# B&R Automation Studio project NAINV104C00R8L515F00 (part 5)

#### fHermesParseBoardAvailable.st
```iecst
(* Hermes Parse XML Table Data For Board Available *)
FUNCTION fHermesParseBoardAvailable

	fHermesParseBoardAvailable	:= TRUE;

	IF (tyXMLTableCurr.sTitle = 'AT') AND (sCurrValueLowerCase = 'boardid') THEN

		p_tyBoardAvailable.tyAvl.bBoardId	:= TRUE;

		IF tyXMLTableNxt.sTitle = 'AV' THEN
			p_tyBoardAvailable.tyData.sBoardId	:= tyXMLTableNxt.sValue;
		END_IF

	ELSIF (tyXMLTableCurr.sTitle = 'AT') AND (sCurrValueLowerCase = 'boardidcreatedby') THEN

		p_tyBoardAvailable.tyAvl.bBoardIdCreatedBy	:= TRUE;

		IF tyXMLTableNxt.sTitle = 'AV' THEN
			p_tyBoardAvailable.tyData.sBoardIdCreatedBy	:= tyXMLTableNxt.sValue;
		END_IF

	ELSIF (tyXMLTableCurr.sTitle = 'AT') AND (sCurrValueLowerCase = 'failedboard') THEN

		p_tyBoardAvailable.tyAvl.bFailedBoard	:= TRUE;

		IF tyXMLTableNxt.sTitle = 'AV' THEN
			IF tyXMLTableNxt.sValue = '1' THEN
				p_tyBoardAvailable.tyData.eFailedBoard	:= HermesGoodBoard;
			ELSIF tyXMLTableNxt.sValue = '2' THEN
				p_tyBoardAvailable.tyData.eFailedBoard	:= HermesFailedBoard;
			ELSE
				p_tyBoardAvailable.tyData.eFailedBoard	:= HermesUnknownBoard;
			END_IF
		END_IF

	ELSIF (tyXMLTableCurr.sTitle = 'AT') AND (sCurrValueLowerCase = 'producttypeid') THEN

		p_tyBoardAvailable.tyAvl.bProductTypeId	:= TRUE;

		IF tyXMLTableNxt.sTitle = 'AV' THEN
			p_tyBoardAvailable.tyData.sProductTypeId	:= tyXMLTableNxt.sValue;
		END_IF

	ELSIF (tyXMLTableCurr.sTitle = 'AT') AND (sCurrValueLowerCase = 'flippedboard') THEN

		p_tyBoardAvailable.tyAvl.bFlippedBoard	:= TRUE;

		IF tyXMLTableNxt.sTitle = 'AV' THEN
			IF tyXMLTableNxt.sValue = '1' THEN
				p_tyBoardAvailable.tyData.eFlippedBoard	:= HermesFlippedBoardTopSideUp;
			ELSIF tyXMLTableNxt.sValue = '2' THEN
				p_tyBoardAvailable.tyData.eFlippedBoard	:= HermesFlippedBoardBtmSideUp;
			ELSE
				p_tyBoardAvailable.tyData.eFlippedBoard	:= HermesFlippedBoardUnknownSide;
			END_IF
		END_IF

	ELSIF (tyXMLTableCurr.sTitle = 'AT') AND (sCurrValueLowerCase = 'topbarcode') THEN

		p_tyBoardAvailable.tyAvl.bTopBarcode	:= TRUE;

		IF tyXMLTableNxt.sTitle = 'AV' THEN
			p_tyBoardAvailable.tyData.sTopBarcode	:= tyXMLTableNxt.sValue;
		END_IF

	ELSIF (tyXMLTableCurr.sTitle = 'AT') AND (sCurrValueLowerCase = 'bottombarcode') THEN

		p_tyBoardAvailable.tyAvl.bBottomBarcode	:= TRUE;

		IF tyXMLTableNxt.sTitle = 'AV' THEN
			p_tyBoardAvailable.tyData.sBottomBarcode	:= tyXMLTableNxt.sValue;
		END_IF

	ELSIF (tyXMLTableCurr.sTitle = 'AT') AND (sCurrValueLowerCase = 'length') THEN

		p_tyBoardAvailable.tyAvl.bLength	:= TRUE;

		IF tyXMLTableNxt.sTitle = 'AV' THEN
			p_tyBoardAvailable.tyData.rLength	:= STRING_TO_REAL(tyXMLTableNxt.sValue);
		END_IF

	ELSIF (tyXMLTableCurr.sTitle = 'AT') AND (sCurrValueLowerCase = 'width') THEN

		p_tyBoardAvailable.tyAvl.bWidth	:= TRUE;

		IF tyXMLTableNxt.sTitle = 'AV' THEN
			p_tyBoardAvailable.tyData.rWidth	:= STRING_TO_REAL(tyXMLTableNxt.sValue);
		END_IF

	ELSIF (tyXMLTableCurr.sTitle = 'AT') AND (sCurrValueLowerCase = 'thickness') THEN

		p_tyBoardAvailable.tyAvl.bThickness	:= TRUE;

		IF tyXMLTableNxt.sTitle = 'AV' THEN
			p_tyBoardAvailable.tyData.rThickness	:= STRING_TO_REAL(tyXMLTableNxt.sValue);
		END_IF

	ELSIF (tyXMLTableCurr.sTitle = 'AT') AND (sCurrValueLowerCase = 'conveyorspeed') THEN

		p_tyBoardAvailable.tyAvl.bConveyorSpeed	:= TRUE;

		IF tyXMLTableNxt.sTitle = 'AV' THEN
			p_tyBoardAvailable.tyData.rConveyorSpeed	:= STRING_TO_REAL(tyXMLTableNxt.sValue);
		END_IF

	ELSIF (tyXMLTableCurr.sTitle = 'AT') AND (sCurrValueLowerCase = 'topclearanceheight') THEN

		p_tyBoardAvailable.tyAvl.bTopClearanceHeight	:= TRUE;

		IF tyXMLTableNxt.sTitle = 'AV' THEN
			p_tyBoardAvailable.tyData.rTopClearanceHeight	:= STRING_TO_REAL(tyXMLTableNxt.sValue);
		END_IF

	ELSIF (tyXMLTableCurr.sTitle = 'AT') AND (sCurrValueLowerCase = 'bottomclearanceheight') THEN

		p_tyBoardAvailable.tyAvl.bBottomClearanceHeight	:= TRUE;

		IF tyXMLTableNxt.sTitle = 'AV' THEN
			p_tyBoardAvailable.tyData.rBottomClearanceHeight	:= STRING_TO_REAL(tyXMLTableNxt.sValue);
		END_IF

	ELSIF (tyXMLTableCurr.sTitle = 'AT') AND (sCurrValueLowerCase = 'weight') THEN

		p_tyBoardAvailable.tyAvl.bWeight	:= TRUE;

		IF tyXMLTableNxt.sTitle = 'AV' THEN
			p_tyBoardAvailable.tyData.rWeight	:= STRING_TO_REAL(tyXMLTableNxt.sValue);
		END_IF

	ELSIF (tyXMLTableCurr.sTitle = 'AT') AND (sCurrValueLowerCase = 'workorderid') THEN

		p_tyBoardAvailable.tyAvl.bWorkOrderId	:= TRUE;

		IF tyXMLTableNxt.sTitle = 'AV' THEN
			p_tyBoardAvailable.tyData.sWorkOrderId	:= tyXMLTableNxt.sValue;
		END_IF

	ELSIF (tyXMLTableCurr.sTitle = 'AT') AND (sCurrValueLowerCase = 'batchid') THEN

		p_tyBoardAvailable.tyAvl.bBatchId	:= TRUE;

		IF tyXMLTableNxt.sTitle = 'AV' THEN
			p_tyBoardAvailable.tyData.sBatchId	:= tyXMLTableNxt.sValue;
		END_IF
	ELSIF (tyXMLTableCurr.sTitle = 'AT') AND (sCurrValueLowerCase = 'route') THEN

		p_tyBoardAvailable.tyAvl.bRoute	:= TRUE;

		IF tyXMLTableNxt.sTitle = 'AV' THEN
			p_tyBoardAvailable.tyData.iRoute	:= STRING_TO_INT(tyXMLTableNxt.sValue);
		END_IF
	ELSIF (tyXMLTableCurr.sTitle = 'AT') AND (sCurrValueLowerCase = 'action') THEN

		p_tyBoardAvailable.tyAvl.bAction	:= TRUE;

		IF tyXMLTableNxt.sTitle = 'AV' THEN
			p_tyBoardAvailable.tyData.iAction	:= STRING_TO_INT(tyXMLTableNxt.sValue);
		END_IF
	ELSIF (tyXMLTableCurr.sTitle = 'ST') AND (sCurrValueLowerCase = 'sb') THEN
		iSubBoardCntr := iSubBoardCntr + 1;
	ELSIF (tyXMLTableCurr.sTitle = 'AT') AND (sCurrValueLowerCase = 'pos') THEN
		p_tyBoardAvailable.tyAvl.tySubBoards.bSubBoardsPos[iSubBoardCntr]	:= TRUE;

		IF tyXMLTableNxt.sTitle = 'AV' THEN
			p_tyBoardAvailable.tyData.tySubBoards.iSubBoardsPos[iSubBoardCntr]	:= STRING_TO_INT(tyXMLTableNxt.sValue);
		END_IF
	ELSIF (tyXMLTableCurr.sTitle = 'AT') AND (sCurrValueLowerCase = 'bc') THEN

		p_tyBoardAvailable.tyAvl.tySubBoards.bSubBoardsBc[iSubBoardCntr]	:= TRUE;

		IF tyXMLTableNxt.sTitle = 'AV' THEN
			p_tyBoardAvailable.tyData.tySubBoards.sSubBoardsBc[iSubBoardCntr]	:= tyXMLTableNxt.sValue;
		END_IF
	ELSIF (tyXMLTableCurr.sTitle = 'AT') AND (sCurrValueLowerCase = 'st') THEN

		p_tyBoardAvailable.tyAvl.tySubBoards.bSubBoardsSt[iSubBoardCntr]	:= TRUE;

		IF tyXMLTableNxt.sTitle = 'AV' THEN
			p_tyBoardAvailable.tyData.tySubBoards.iSubBoardsSt[iSubBoardCntr]	:= STRING_TO_INT(tyXMLTableNxt.sValue);
		END_IF
	END_IF

END_FUNCTION
```

#### fHermesParseMachineReady.st
```iecst
(* Hermes Parse XML Table Data For Machine Ready*)
FUNCTION fHermesParseMachineReady

	fHermesParseMachineReady	:= TRUE;

	IF (tyXMLTableCurr.sTitle = 'AT') AND (sCurrValueLowerCase = 'failedboard') THEN

		p_tyMachineReady.tyAvl.bFailedBoard	:= TRUE;

		IF tyXMLTableNxt.sTitle = 'AV' THEN
			IF tyXMLTableNxt.sValue = '1' THEN
				p_tyMachineReady.tyData.eFailedBoard	:= HermesGoodBoard;
			ELSIF tyXMLTableNxt.sValue = '2' THEN
				p_tyMachineReady.tyData.eFailedBoard	:= HermesFailedBoard;
			ELSE
				p_tyMachineReady.tyData.eFailedBoard	:= HermesUnknownBoard;
			END_IF
		END_IF

	ELSIF (tyXMLTableCurr.sTitle = 'AT') AND (sCurrValueLowerCase = 'forecastid') THEN

		p_tyMachineReady.tyAvl.bForecastId	:= TRUE;

		IF tyXMLTableNxt.sTitle = 'AV' THEN
			p_tyMachineReady.tyData.sForecastId	:= tyXMLTableNxt.sValue;
		END_IF

	ELSIF (tyXMLTableCurr.sTitle = 'AT') AND (sCurrValueLowerCase = 'boardid') THEN

		p_tyMachineReady.tyAvl.bBoardId	:= TRUE;

		IF tyXMLTableNxt.sTitle = 'AV' THEN
			p_tyMachineReady.tyData.sBoardId	:= tyXMLTableNxt.sValue;
		END_IF

	ELSIF (tyXMLTableCurr.sTitle = 'AT') AND (sCurrValueLowerCase = 'producttypeid') THEN

		p_tyMachineReady.tyAvl.bProductTypeId	:= TRUE;

		IF tyXMLTableNxt.sTitle = 'AV' THEN
			p_tyMachineReady.tyData.sProductTypeId	:= tyXMLTableNxt.sValue;
		END_IF

	ELSIF (tyXMLTableCurr.sTitle = 'AT') AND (sCurrValueLowerCase = 'flippedboard') THEN

		p_tyMachineReady.tyAvl.bFlippedBoard	:= TRUE;

		IF tyXMLTableNxt.sTitle = 'AV' THEN
			IF tyXMLTableNxt.sValue = '1' THEN
				p_tyMachineReady.tyData.eFlippedBoard	:= HermesFlippedBoardTopSideUp;
			ELSIF tyXMLTableNxt.sValue = '2' THEN
				p_tyMachineReady.tyData.eFlippedBoard	:= HermesFlippedBoardBtmSideUp;
			ELSE
				p_tyMachineReady.tyData.eFlippedBoard	:= HermesFlippedBoardUnknownSide;
			END_IF
		END_IF

	ELSIF (tyXMLTableCurr.sTitle = 'AT') AND (sCurrValueLowerCase = 'length') THEN

		p_tyMachineReady.tyAvl.bLength	:= TRUE;

		IF tyXMLTableNxt.sTitle = 'AV' THEN
			p_tyMachineReady.tyData.rLength	:= STRING_TO_REAL(tyXMLTableNxt.sValue);
		END_IF

	ELSIF (tyXMLTableCurr.sTitle = 'AT') AND (sCurrValueLowerCase = 'width') THEN

		p_tyMachineReady.tyAvl.bWidth	:= TRUE;

		IF tyXMLTableNxt.sTitle = 'AV' THEN
			p_tyMachineReady.tyData.rWidth	:= STRING_TO_REAL(tyXMLTableNxt.sValue);
		END_IF

	ELSIF (tyXMLTableCurr.sTitle = 'AT') AND (sCurrValueLowerCase = 'thickness') THEN

		p_tyMachineReady.tyAvl.bThickness	:= TRUE;

		IF tyXMLTableNxt.sTitle = 'AV' THEN
			p_tyMachineReady.tyData.rThickness	:= STRING_TO_REAL(tyXMLTableNxt.sValue);
		END_IF

	ELSIF (tyXMLTableCurr.sTitle = 'AT') AND (sCurrValueLowerCase = 'conveyorspeed') THEN

		p_tyMachineReady.tyAvl.bConveyorSpeed	:= TRUE;

		IF tyXMLTableNxt.sTitle = 'AV' THEN
			p_tyMachineReady.tyData.rConveyorSpeed	:= STRING_TO_REAL(tyXMLTableNxt.sValue);
		END_IF

	ELSIF (tyXMLTableCurr.sTitle = 'AT') AND (sCurrValueLowerCase = 'topclearanceheight') THEN

		p_tyMachineReady.tyAvl.bTopClearanceHeight	:= TRUE;

		IF tyXMLTableNxt.sTitle = 'AV' THEN
			p_tyMachineReady.tyData.rTopClearanceHeight	:= STRING_TO_REAL(tyXMLTableNxt.sValue);
		END_IF

	ELSIF (tyXMLTableCurr.sTitle = 'AT') AND (sCurrValueLowerCase = 'bottomclearanceheight') THEN

		p_tyMachineReady.tyAvl.bBottomClearanceHeight	:= TRUE;

		IF tyXMLTableNxt.sTitle = 'AV' THEN
			p_tyMachineReady.tyData.rBottomClearanceHeight	:= STRING_TO_REAL(tyXMLTableNxt.sValue);
		END_IF

	ELSIF (tyXMLTableCurr.sTitle = 'AT') AND (sCurrValueLowerCase = 'weight') THEN

		p_tyMachineReady.tyAvl.bWeight	:= TRUE;

		IF tyXMLTableNxt.sTitle = 'AV' THEN
			p_tyMachineReady.tyData.rWeight	:= STRING_TO_REAL(tyXMLTableNxt.sValue);
		END_IF

	ELSIF (tyXMLTableCurr.sTitle = 'AT') AND (sCurrValueLowerCase = 'workorderid') THEN

		p_tyMachineReady.tyAvl.bWorkOrderId	:= TRUE;

		IF tyXMLTableNxt.sTitle = 'AV' THEN
			p_tyMachineReady.tyData.sWorkOrderId	:= tyXMLTableNxt.sValue;
		END_IF

	ELSIF (tyXMLTableCurr.sTitle = 'AT') AND (sCurrValueLowerCase = 'batchid') THEN

		p_tyMachineReady.tyAvl.bBatchId	:= TRUE;

		IF tyXMLTableNxt.sTitle = 'AV' THEN
			p_tyMachineReady.tyData.sBatchId	:= tyXMLTableNxt.sValue;
		END_IF

	END_IF

END_FUNCTION
```

#### fHermesParseStartTransport.st
```iecst
(* Hermes Parse XML Table Data For Start Transport*)
FUNCTION fHermesParseStartTransport

	fHermesParseStartTransport	:= TRUE;

	IF (tyXMLTableCurr.sTitle = 'AT') AND (sCurrValueLowerCase = 'boardid') THEN

		p_tyStartTransport.tyAvl.bBoardId	:= TRUE;

		IF tyXMLTableNxt.sTitle = 'AV' THEN
			p_tyStartTransport.tyData.sBoardId	:= tyXMLTableNxt.sValue;
		END_IF

	ELSIF (tyXMLTableCurr.sTitle = 'AT') AND (sCurrValueLowerCase = 'conveyorspeed') THEN

		p_tyStartTransport.tyAvl.bConveyorSpeed	:= TRUE;

		IF tyXMLTableNxt.sTitle = 'AV' THEN
			p_tyStartTransport.tyData.rConveyorSpeed	:= STRING_TO_REAL(tyXMLTableNxt.sValue);
		END_IF

	END_IF

END_FUNCTION
```

#### fHermesParseStopTransport.st
```iecst
(* Hermes Parse XML Table Data For Stop Transport*)
FUNCTION fHermesParseStopTransport

	fHermesParseStopTransport	:= TRUE;

	IF (tyXMLTableCurr.sTitle = 'AT') AND (sCurrValueLowerCase = 'transferstate') THEN

		p_tyStopTransport.tyAvl.bTransferState	:= TRUE;

		IF tyXMLTableNxt.sTitle = 'AV' THEN
			IF tyXMLTableNxt.sValue = '1' THEN
				p_tyStopTransport.tyData.eTransferState	:= HermesTransferStateNotStarted;
			ELSIF tyXMLTableNxt.sValue = '2' THEN
				p_tyStopTransport.tyData.eTransferState	:= HermesTransferStateIncomplete;
			ELSE
				p_tyStopTransport.tyData.eTransferState	:= HermesTransferStateComplete;
			END_IF
		END_IF

	ELSIF (tyXMLTableCurr.sTitle = 'AT') AND (sCurrValueLowerCase = 'boardid') THEN

		p_tyStopTransport.tyAvl.bBoardId	:= TRUE;

		IF tyXMLTableNxt.sTitle = 'AV' THEN
			p_tyStopTransport.tyData.sBoardId	:= tyXMLTableNxt.sValue;
		END_IF

	END_IF

END_FUNCTION
```

#### fHermesParseTransportFinished.st
```iecst
(* Hermes Parse XML Table Data For Transport Finished *)
FUNCTION fHermesParseTransportFinished

	fHermesParseTransportFinished	:= TRUE;

	IF (tyXMLTableCurr.sTitle = 'AT') AND (sCurrValueLowerCase = 'transferstate') THEN

		p_tyTransportFinished.tyAvl.bTransferState	:= TRUE;

		IF tyXMLTableNxt.sTitle = 'AV' THEN
			IF tyXMLTableNxt.sValue = '1' THEN
				p_tyTransportFinished.tyData.eTransferState	:= HermesTransferStateNotStarted;
			ELSIF tyXMLTableNxt.sValue = '2' THEN
				p_tyTransportFinished.tyData.eTransferState	:= HermesTransferStateIncomplete;
			ELSE
				p_tyTransportFinished.tyData.eTransferState	:= HermesTransferStateComplete;
			END_IF
		END_IF

	ELSIF (tyXMLTableCurr.sTitle = 'AT') AND (sCurrValueLowerCase = 'boardid') THEN

		p_tyTransportFinished.tyAvl.bBoardId	:= TRUE;

		IF tyXMLTableNxt.sTitle = 'AV' THEN
			p_tyTransportFinished.tyData.sBoardId	:= tyXMLTableNxt.sValue;
		END_IF

	END_IF

END_FUNCTION
```

#### fHermesParseSetConfiguration.st
```iecst
(* Hermes Parse XML Table Data For Set Configuration*)
FUNCTION fHermesParseSetConfiguration

	fHermesParseSetConfiguration	:= TRUE;

	IF (tyXMLTableCurr.sTitle = 'AT') AND (sCurrValueLowerCase = 'machineid') THEN

		p_tySetConfiguration.tyAvl.bMachineId	:= TRUE;

		IF tyXMLTableNxt.sTitle = 'AV' THEN
			p_tySetConfiguration.tyData.sMachineId	:= tyXMLTableNxt.sValue;
		END_IF

	ELSIF (tyXMLTableCurr.sTitle = 'AT') AND (sCurrValueLowerCase = 'supervisorysystemport') THEN

		p_tySetConfiguration.tyAvl.bSupervisorySystemPort	:= TRUE;

		IF tyXMLTableNxt.sTitle = 'AV' THEN
			p_tySetConfiguration.tyData.uiSupervisorySystemPort	:= STRING_TO_UINT(tyXMLTableNxt.sValue);
		END_IF

	ELSIF (tyXMLTableCurr.sTitle = 'ST') AND (sCurrValueLowerCase = 'upstreamconfigurations') THEN

		bUpstream	:= TRUE;
		bDownstream	:= FALSE;

	ELSIF (tyXMLTableCurr.sTitle = 'ET') AND (sCurrValueLowerCase = 'upstreamconfigurations') THEN

		bUpstream	:= FALSE;

	ELSIF (tyXMLTableCurr.sTitle = 'ST') AND (sCurrValueLowerCase = 'downstreamconfigurations') THEN

		bUpstream	:= FALSE;
		bDownstream	:= TRUE;

	ELSIF (tyXMLTableCurr.sTitle = 'ET') AND (sCurrValueLowerCase = 'downstreamconfigurations') THEN

		bDownstream	:= FALSE;

	ELSIF bUpstream = TRUE THEN

		IF (tyXMLTableCurr.sTitle = 'ST') AND (sCurrValueLowerCase = 'upstreamconfiguration') THEN

			p_tySetConfiguration.tyAvl.bUpstreamConfigurations	:= TRUE;

			p_tySetConfiguration.tyAvl.iUpstreamConfigurations	:= p_tySetConfiguration.tyAvl.iUpstreamConfigurations + 1;
//			IF p_tySetConfiguration.tyAvl.iUpstreamConfigurations > 3 THEN
//				p_tySetConfiguration.tyAvl.iUpstreamConfigurations	:= 3;
//			END_IF

		ELSIF p_tySetConfiguration.tyAvl.iUpstreamConfigurations <> 0 THEN

			IF (tyXMLTableCurr.sTitle = 'AT') AND (sCurrValueLowerCase = 'upstreamlaneid') THEN

				p_tySetConfiguration.tyAvl.a_tyUpstreamConfigurations[p_tySetConfiguration.tyAvl.iUpstreamConfigurations - 1].bUpstreamLaneId	:= TRUE;

				IF tyXMLTableNxt.sTitle = 'AV' THEN
					p_tySetConfiguration.tyData.a_tyUpstreamConfigurations[p_tySetConfiguration.tyAvl.iUpstreamConfigurations - 1].iUpstreamLaneId	:= STRING_TO_INT(tyXMLTableNxt.sValue);
				END_IF

			ELSIF (tyXMLTableCurr.sTitle = 'AT') AND (sCurrValueLowerCase = 'upstreaminterfaceid') THEN

				p_tySetConfiguration.tyAvl.a_tyUpstreamConfigurations[p_tySetConfiguration.tyAvl.iUpstreamConfigurations - 1].bUpstreamInterfaceId	:= TRUE;

				IF tyXMLTableNxt.sTitle = 'AV' THEN
					p_tySetConfiguration.tyData.a_tyUpstreamConfigurations[p_tySetConfiguration.tyAvl.iUpstreamConfigurations - 1].sUpstreamInterfaceId	:= tyXMLTableNxt.sValue;
				END_IF

			ELSIF (tyXMLTableCurr.sTitle = 'AT') AND (sCurrValueLowerCase = 'hostaddress') THEN

				p_tySetConfiguration.tyAvl.a_tyUpstreamConfigurations[p_tySetConfiguration.tyAvl.iUpstreamConfigurations - 1].bHostAddress	:= TRUE;

				IF tyXMLTableNxt.sTitle = 'AV' THEN
					p_tySetConfiguration.tyData.a_tyUpstreamConfigurations[p_tySetConfiguration.tyAvl.iUpstreamConfigurations - 1].sHostAddress	:= tyXMLTableNxt.sValue;
				END_IF

			ELSIF (tyXMLTableCurr.sTitle = 'AT') AND (sCurrValueLowerCase = 'port') THEN

				p_tySetConfiguration.tyAvl.a_tyUpstreamConfigurations[p_tySetConfiguration.tyAvl.iUpstreamConfigurations - 1].bPort	:= TRUE;

				IF tyXMLTableNxt.sTitle = 'AV' THEN
					p_tySetConfiguration.tyData.a_tyUpstreamConfigurations[p_tySetConfiguration.tyAvl.iUpstreamConfigurations - 1].uiPort	:= STRING_TO_UINT(tyXMLTableNxt.sValue);
				END_IF

			END_IF

		END_IF

	ELSIF bDownstream = TRUE THEN

		IF (tyXMLTableCurr.sTitle = 'ST') AND (sCurrValueLowerCase = 'downstreamconfiguration') THEN

			p_tySetConfiguration.tyAvl.bDownstreamConfigurations	:= TRUE;

			p_tySetConfiguration.tyAvl.iDownstreamConfigurations	:= p_tySetConfiguration.tyAvl.iDownstreamConfigurations + 1;
//			IF p_tySetConfiguration.tyAvl.iDownstreamConfigurations > 3 THEN
//				p_tySetConfiguration.tyAvl.iDownstreamConfigurations	:= 3;
//			END_IF

		ELSIF p_tySetConfiguration.tyAvl.iDownstreamConfigurations <> 0 THEN

			IF (tyXMLTableCurr.sTitle = 'AT') AND (sCurrValueLowerCase = 'downstreamlaneid') THEN

				p_tySetConfiguration.tyAvl.a_tyDownstreamConfigurations[p_tySetConfiguration.tyAvl.iDownstreamConfigurations - 1].bDownstreamLaneId	:= TRUE;

				IF tyXMLTableNxt.sTitle = 'AV' THEN
					p_tySetConfiguration.tyData.a_tyDownstreamConfigurations[p_tySetConfiguration.tyAvl.iDownstreamConfigurations - 1].iDownstreamLaneId	:= STRING_TO_INT(tyXMLTableNxt.sValue);
				END_IF

			ELSIF (tyXMLTableCurr.sTitle = 'AT') AND (sCurrValueLowerCase = 'downstreaminterfaceid') THEN

				p_tySetConfiguration.tyAvl.a_tyDownstreamConfigurations[p_tySetConfiguration.tyAvl.iDownstreamConfigurations - 1].bDownstreamInterfaceId	:= TRUE;

				IF tyXMLTableNxt.sTitle = 'AV' THEN
					p_tySetConfiguration.tyData.a_tyDownstreamConfigurations[p_tySetConfiguration.tyAvl.iDownstreamConfigurations - 1].sDownstreamInterfaceId	:= tyXMLTableNxt.sValue;
				END_IF

			ELSIF (tyXMLTableCurr.sTitle = 'AT') AND (sCurrValueLowerCase = 'clientaddress') THEN

				p_tySetConfiguration.tyAvl.a_tyDownstreamConfigurations[p_tySetConfiguration.tyAvl.iDownstreamConfigurations - 1].bClientAddress	:= TRUE;

				IF tyXMLTableNxt.sTitle = 'AV' THEN
					p_tySetConfiguration.tyData.a_tyDownstreamConfigurations[p_tySetConfiguration.tyAvl.iDownstreamConfigurations - 1].sClientAddress	:= tyXMLTableNxt.sValue;
				END_IF

			ELSIF (tyXMLTableCurr.sTitle = 'AT') AND (sCurrValueLowerCase = 'port') THEN

				p_tySetConfiguration.tyAvl.a_tyDownstreamConfigurations[p_tySetConfiguration.tyAvl.iDownstreamConfigurations - 1].bPort	:= TRUE;

				IF tyXMLTableNxt.sTitle = 'AV' THEN
					p_tySetConfiguration.tyData.a_tyDownstreamConfigurations[p_tySetConfiguration.tyAvl.iDownstreamConfigurations - 1].uiPort	:= STRING_TO_UINT(tyXMLTableNxt.sValue);
				END_IF

			END_IF

		END_IF

	END_IF

END_FUNCTION
```

#### fHermesParseCurrentConfiguration.st
```iecst
(* Hermes Parse XML Table Data For Current Configuration*)
FUNCTION fHermesParseCurrentConfiguration

	fHermesParseCurrentConfiguration	:= TRUE;

	IF (tyXMLTableCurr.sTitle = 'AT') AND (sCurrValueLowerCase = 'machineid') THEN

		p_tyCurrentConfiguration.tyAvl.bMachineId	:= TRUE;

		IF tyXMLTableNxt.sTitle = 'AV' THEN
			p_tyCurrentConfiguration.tyData.sMachineId	:= tyXMLTableNxt.sValue;
		END_IF

	ELSIF (tyXMLTableCurr.sTitle = 'AT') AND (sCurrValueLowerCase = 'supervisorysytemport') THEN

			p_tyCurrentConfiguration.tyAvl.bSupervisorySystemPort	:= TRUE;

			IF tyXMLTableNxt.sTitle = 'AV' THEN
				p_tyCurrentConfiguration.tyData.uiSupervisorySystemPort	:= STRING_TO_UINT(tyXMLTableNxt.sValue);
			END_IF

	ELSIF (tyXMLTableCurr.sTitle = 'ST') AND (sCurrValueLowerCase = 'upstreamconfigurations') THEN

		bUpstream	:= TRUE;
		bDownstream	:= FALSE;

	ELSIF (tyXMLTableCurr.sTitle = 'ET') AND (sCurrValueLowerCase = 'upstreamconfigurations') THEN

		bUpstream	:= FALSE;

	ELSIF (tyXMLTableCurr.sTitle = 'ST') AND (sCurrValueLowerCase = 'downstreamconfigurations') THEN

		bUpstream	:= FALSE;
		bDownstream	:= TRUE;

	ELSIF (tyXMLTableCurr.sTitle = 'ET') AND (sCurrValueLowerCase = 'downstreamconfigurations') THEN

		bDownstream	:= FALSE;

	ELSIF bUpstream = TRUE THEN

		IF (tyXMLTableCurr.sTitle = 'ST') AND (sCurrValueLowerCase = 'upstreamconfiguration') THEN

			p_tyCurrentConfiguration.tyAvl.bUpstreamConfigurations	:= TRUE;

			p_tyCurrentConfiguration.tyAvl.iUpstreamConfigurations	:= p_tyCurrentConfiguration.tyAvl.iUpstreamConfigurations + 1;
			IF p_tyCurrentConfiguration.tyAvl.iUpstreamConfigurations > 3 THEN
				p_tyCurrentConfiguration.tyAvl.iUpstreamConfigurations	:= 3;
			END_IF

		ELSIF p_tyCurrentConfiguration.tyAvl.iUpstreamConfigurations <> 0 THEN

			IF (tyXMLTableCurr.sTitle = 'AT') AND (sCurrValueLowerCase = 'upstreamlaneid') THEN

				p_tyCurrentConfiguration.tyAvl.a_tyUpstreamConfigurations[p_tyCurrentConfiguration.tyAvl.iUpstreamConfigurations - 1].bUpstreamLaneId	:= TRUE;

				IF tyXMLTableNxt.sTitle = 'AV' THEN
					p_tyCurrentConfiguration.tyData.a_tyUpstreamConfigurations[p_tyCurrentConfiguration.tyAvl.iUpstreamConfigurations - 1].iUpstreamLaneId	:= STRING_TO_INT(tyXMLTableNxt.sValue);
				END_IF

			ELSIF (tyXMLTableCurr.sTitle = 'AT') AND (sCurrValueLowerCase = 'upstreaminterfaceid') THEN

				p_tyCurrentConfiguration.tyAvl.a_tyUpstreamConfigurations[p_tyCurrentConfiguration.tyAvl.iUpstreamConfigurations - 1].bUpstreamInterfaceId	:= TRUE;

				IF tyXMLTableNxt.sTitle = 'AV' THEN
					p_tyCurrentConfiguration.tyData.a_tyUpstreamConfigurations[p_tyCurrentConfiguration.tyAvl.iUpstreamConfigurations - 1].sUpstreamInterfaceId	:= tyXMLTableNxt.sValue;
				END_IF

			ELSIF (tyXMLTableCurr.sTitle = 'AT') AND (sCurrValueLowerCase = 'hostaddress') THEN

				p_tyCurrentConfiguration.tyAvl.a_tyUpstreamConfigurations[p_tyCurrentConfiguration.tyAvl.iUpstreamConfigurations - 1].bHostAddress	:= TRUE;

				IF tyXMLTableNxt.sTitle = 'AV' THEN
					p_tyCurrentConfiguration.tyData.a_tyUpstreamConfigurations[p_tyCurrentConfiguration.tyAvl.iUpstreamConfigurations - 1].sHostAddress	:= tyXMLTableNxt.sValue;
				END_IF

			ELSIF (tyXMLTableCurr.sTitle = 'AT') AND (sCurrValueLowerCase = 'port') THEN

				p_tyCurrentConfiguration.tyAvl.a_tyUpstreamConfigurations[p_tyCurrentConfiguration.tyAvl.iUpstreamConfigurations - 1].bPort	:= TRUE;

				IF tyXMLTableNxt.sTitle = 'AV' THEN
					p_tyCurrentConfiguration.tyData.a_tyUpstreamConfigurations[p_tyCurrentConfiguration.tyAvl.iUpstreamConfigurations - 1].uiPort	:= STRING_TO_UINT(tyXMLTableNxt.sValue);
				END_IF

			END_IF

		END_IF

	ELSIF bDownstream = TRUE THEN

		IF (tyXMLTableCurr.sTitle = 'ST') AND (sCurrValueLowerCase = 'downstreamconfiguration') THEN

			p_tyCurrentConfiguration.tyAvl.bDownstreamConfigurations	:= TRUE;

			p_tyCurrentConfiguration.tyAvl.iDownstreamConfigurations	:= p_tyCurrentConfiguration.tyAvl.iDownstreamConfigurations + 1;
			IF p_tyCurrentConfiguration.tyAvl.iDownstreamConfigurations > 3 THEN
				p_tyCurrentConfiguration.tyAvl.iDownstreamConfigurations	:= 3;
			END_IF

		ELSIF p_tyCurrentConfiguration.tyAvl.iDownstreamConfigurations <> 0 THEN

			IF (tyXMLTableCurr.sTitle = 'AT') AND (sCurrValueLowerCase = 'downstreamlaneid') THEN

				p_tyCurrentConfiguration.tyAvl.a_tyDownstreamConfigurations[p_tyCurrentConfiguration.tyAvl.iDownstreamConfigurations - 1].bDownstreamLaneId	:= TRUE;

				IF tyXMLTableNxt.sTitle = 'AV' THEN
					p_tyCurrentConfiguration.tyData.a_tyDownstreamConfigurations[p_tyCurrentConfiguration.tyAvl.iDownstreamConfigurations - 1].iDownstreamLaneId	:= STRING_TO_INT(tyXMLTableNxt.sValue);
				END_IF

			ELSIF (tyXMLTableCurr.sTitle = 'AT') AND (sCurrValueLowerCase = 'downstreaminterfaceid') THEN

				p_tyCurrentConfiguration.tyAvl.a_tyDownstreamConfigurations[p_tyCurrentConfiguration.tyAvl.iDownstreamConfigurations - 1].bDownstreamInterfaceId	:= TRUE;

				IF tyXMLTableNxt.sTitle = 'AV' THEN
					p_tyCurrentConfiguration.tyData.a_tyDownstreamConfigurations[p_tyCurrentConfiguration.tyAvl.iDownstreamConfigurations - 1].sDownstreamInterfaceId	:= tyXMLTableNxt.sValue;
				END_IF

			ELSIF (tyXMLTableCurr.sTitle = 'AT') AND (sCurrValueLowerCase = 'clientaddress') THEN

				p_tyCurrentConfiguration.tyAvl.a_tyDownstreamConfigurations[p_tyCurrentConfiguration.tyAvl.iDownstreamConfigurations - 1].bClientAddress	:= TRUE;

				IF tyXMLTableNxt.sTitle = 'AV' THEN
					p_tyCurrentConfiguration.tyData.a_tyDownstreamConfigurations[p_tyCurrentConfiguration.tyAvl.iDownstreamConfigurations - 1].sClientAddress	:= tyXMLTableNxt.sValue;
				END_IF

			ELSIF (tyXMLTableCurr.sTitle = 'AT') AND (sCurrValueLowerCase = 'port') THEN

				p_tyCurrentConfiguration.tyAvl.a_tyDownstreamConfigurations[p_tyCurrentConfiguration.tyAvl.iDownstreamConfigurations - 1].bPort	:= TRUE;

				IF tyXMLTableNxt.sTitle = 'AV' THEN
					p_tyCurrentConfiguration.tyData.a_tyDownstreamConfigurations[p_tyCurrentConfiguration.tyAvl.iDownstreamConfigurations - 1].uiPort	:= STRING_TO_UINT(tyXMLTableNxt.sValue);
				END_IF

			END_IF

		END_IF

	END_IF

END_FUNCTION
```

#### fHermesParseBoardForecast.st
```iecst
(* Hermes Parse XML Table Data For Board Forecast*)
FUNCTION fHermesParseBoardForecast

	fHermesParseBoardForecast	:= TRUE;

	IF (tyXMLTableCurr.sTitle = 'AT') AND (sCurrValueLowerCase = 'forecastid') THEN

		p_tyBoardForecast.tyAvl.bForecastId	:= TRUE;

		IF tyXMLTableNxt.sTitle = 'AV' THEN
			p_tyBoardForecast.tyData.sForecastId	:= tyXMLTableNxt.sValue;
		END_IF

	ELSIF (tyXMLTableCurr.sTitle = 'AT') AND (sCurrValueLowerCase = 'timeuntilavailable') THEN

		p_tyBoardForecast.tyAvl.bTimeUntilAvailable	:= TRUE;

		IF tyXMLTableNxt.sTitle = 'AV' THEN
			p_tyBoardForecast.tyData.rTimeUntilAvailable	:= STRING_TO_REAL(tyXMLTableNxt.sValue);
		END_IF

	ELSIF (tyXMLTableCurr.sTitle = 'AT') AND (sCurrValueLowerCase = 'boardid') THEN

		p_tyBoardForecast.tyAvl.bBoardId	:= TRUE;

		IF tyXMLTableNxt.sTitle = 'AV' THEN
			p_tyBoardForecast.tyData.sBoardId	:= tyXMLTableNxt.sValue;
		END_IF

	ELSIF (tyXMLTableCurr.sTitle = 'AT') AND (sCurrValueLowerCase = 'boardidcreatedby') THEN

		p_tyBoardForecast.tyAvl.bBoardIdCreatedBy	:= TRUE;

		IF tyXMLTableNxt.sTitle = 'AV' THEN
			p_tyBoardForecast.tyData.sBoardIdCreatedBy	:= tyXMLTableNxt.sValue;
		END_IF

	ELSIF (tyXMLTableCurr.sTitle = 'AT') AND (sCurrValueLowerCase = 'failedboard') THEN

		p_tyBoardForecast.tyAvl.bFailedBoard	:= TRUE;

		IF tyXMLTableNxt.sTitle = 'AV' THEN
			IF tyXMLTableNxt.sValue = '1' THEN
				p_tyBoardForecast.tyData.eFailedBoard	:= HermesGoodBoard;
			ELSIF tyXMLTableNxt.sValue = '2' THEN
				p_tyBoardForecast.tyData.eFailedBoard	:= HermesFailedBoard;
			ELSE
				p_tyBoardForecast.tyData.eFailedBoard	:= HermesUnknownBoard;
			END_IF
		END_IF

	ELSIF (tyXMLTableCurr.sTitle = 'AT') AND (sCurrValueLowerCase = 'producttypeid') THEN

		p_tyBoardForecast.tyAvl.bProductTypeId	:= TRUE;

		IF tyXMLTableNxt.sTitle = 'AV' THEN
			p_tyBoardForecast.tyData.sProductTypeId	:= tyXMLTableNxt.sValue;
		END_IF

	ELSIF (tyXMLTableCurr.sTitle = 'AT') AND (sCurrValueLowerCase = 'flippedboard') THEN

		p_tyBoardForecast.tyAvl.bFlippedBoard	:= TRUE;

		IF tyXMLTableNxt.sTitle = 'AV' THEN
			IF tyXMLTableNxt.sValue = '1' THEN
				p_tyBoardForecast.tyData.eFlippedBoard	:= HermesFlippedBoardTopSideUp;
			ELSIF tyXMLTableNxt.sValue = '2' THEN
				p_tyBoardForecast.tyData.eFlippedBoard	:= HermesFlippedBoardBtmSideUp;
			ELSE
				p_tyBoardForecast.tyData.eFlippedBoard	:= HermesFlippedBoardUnknownSide;
			END_IF
		END_IF

	ELSIF (tyXMLTableCurr.sTitle = 'AT') AND (sCurrValueLowerCase = 'topbarcode') THEN

		p_tyBoardForecast.tyAvl.bTopBarcode	:= TRUE;

		IF tyXMLTableNxt.sTitle = 'AV' THEN
			p_tyBoardForecast.tyData.sTopBarcode	:= tyXMLTableNxt.sValue;
		END_IF

	ELSIF (tyXMLTableCurr.sTitle = 'AT') AND (sCurrValueLowerCase = 'bottombarcode') THEN

		p_tyBoardForecast.tyAvl.bBottomBarcode	:= TRUE;

		IF tyXMLTableNxt.sTitle = 'AV' THEN
			p_tyBoardForecast.tyData.sBottomBarcode	:= tyXMLTableNxt.sValue;
		END_IF

	ELSIF (tyXMLTableCurr.sTitle = 'AT') AND (sCurrValueLowerCase = 'length') THEN

		p_tyBoardForecast.tyAvl.bLength	:= TRUE;

		IF tyXMLTableNxt.sTitle = 'AV' THEN
			p_tyBoardForecast.tyData.rLength	:= STRING_TO_REAL(tyXMLTableNxt.sValue);
		END_IF

	ELSIF (tyXMLTableCurr.sTitle = 'AT') AND (sCurrValueLowerCase = 'width') THEN

		p_tyBoardForecast.tyAvl.bWidth	:= TRUE;

		IF tyXMLTableNxt.sTitle = 'AV' THEN
			p_tyBoardForecast.tyData.rWidth	:= STRING_TO_REAL(tyXMLTableNxt.sValue);
		END_IF

	ELSIF (tyXMLTableCurr.sTitle = 'AT') AND (sCurrValueLowerCase = 'thickness') THEN

		p_tyBoardForecast.tyAvl.bThickness	:= TRUE;

		IF tyXMLTableNxt.sTitle = 'AV' THEN
			p_tyBoardForecast.tyData.rThickness	:= STRING_TO_REAL(tyXMLTableNxt.sValue);
		END_IF

	ELSIF (tyXMLTableCurr.sTitle = 'AT') AND (sCurrValueLowerCase = 'conveyorspeed') THEN

		p_tyBoardForecast.tyAvl.bConveyorSpeed	:= TRUE;

		IF tyXMLTableNxt.sTitle = 'AV' THEN
			p_tyBoardForecast.tyData.rConveyorSpeed	:= STRING_TO_REAL(tyXMLTableNxt.sValue);
		END_IF

	ELSIF (tyXMLTableCurr.sTitle = 'AT') AND (sCurrValueLowerCase = 'topclearanceheight') THEN

		p_tyBoardForecast.tyAvl.bTopClearanceHeight	:= TRUE;

		IF tyXMLTableNxt.sTitle = 'AV' THEN
			p_tyBoardForecast.tyData.rTopClearanceHeight	:= STRING_TO_REAL(tyXMLTableNxt.sValue);
		END_IF

	ELSIF (tyXMLTableCurr.sTitle = 'AT') AND (sCurrValueLowerCase = 'bottomclearanceheight') THEN

		p_tyBoardForecast.tyAvl.bBottomClearanceHeight	:= TRUE;

		IF tyXMLTableNxt.sTitle = 'AV' THEN
			p_tyBoardForecast.tyData.rBottomClearanceHeight	:= STRING_TO_REAL(tyXMLTableNxt.sValue);
		END_IF

	ELSIF (tyXMLTableCurr.sTitle = 'AT') AND (sCurrValueLowerCase = 'weight') THEN

		p_tyBoardForecast.tyAvl.bWeight	:= TRUE;

		IF tyXMLTableNxt.sTitle = 'AV' THEN
			p_tyBoardForecast.tyData.rWeight	:= STRING_TO_REAL(tyXMLTableNxt.sValue);
		END_IF

	ELSIF (tyXMLTableCurr.sTitle = 'AT') AND (sCurrValueLowerCase = 'workorderid') THEN

		p_tyBoardForecast.tyAvl.bWorkOrderId	:= TRUE;

		IF tyXMLTableNxt.sTitle = 'AV' THEN
			p_tyBoardForecast.tyData.sWorkOrderId	:= tyXMLTableNxt.sValue;
		END_IF

	ELSIF (tyXMLTableCurr.sTitle = 'AT') AND (sCurrValueLowerCase = 'batchid') THEN

		p_tyBoardForecast.tyAvl.bBatchId	:= TRUE;

		IF tyXMLTableNxt.sTitle = 'AV' THEN
			p_tyBoardForecast.tyData.sBatchId	:= tyXMLTableNxt.sValue;
		END_IF

	END_IF

END_FUNCTION
```

#### fHermesParseQueryBoardInfo.st
```iecst
(* Hermes Parse XML Table Data For Query Board Info *)
FUNCTION fHermesParseQueryBoardInfo

	fHermesParseQueryBoardInfo	:= TRUE;

	IF (tyXMLTableCurr.sTitle = 'AT') AND (sCurrValueLowerCase = 'topbarcode') THEN

		p_tyQueryBoardInfo.tyAvl.bTopBarcode	:= TRUE;

		IF tyXMLTableNxt.sTitle = 'AV' THEN
			p_tyQueryBoardInfo.tyData.sTopBarcode	:= tyXMLTableNxt.sValue;
		END_IF

	ELSIF (tyXMLTableCurr.sTitle = 'AT') AND (sCurrValueLowerCase = 'bottombarcode') THEN

		p_tyQueryBoardInfo.tyAvl.bBottomBarcode	:= TRUE;

		IF tyXMLTableNxt.sTitle = 'AV' THEN
			p_tyQueryBoardInfo.tyData.sBottomBarcode	:= tyXMLTableNxt.sValue;
		END_IF

	END_IF

END_FUNCTION
```

#### fHermesParseSendBoardInfo.st
```iecst
(* Hermes Parse XML Table Data For Send Board Info*)
FUNCTION fHermesParseSendBoardInfo

	fHermesParseSendBoardInfo	:= TRUE;

	IF (tyXMLTableCurr.sTitle = 'AT') AND (sCurrValueLowerCase = 'boardid') THEN

		p_tySendBoardInfo.tyAvl.bBoardId	:= TRUE;

		IF tyXMLTableNxt.sTitle = 'AV' THEN
			p_tySendBoardInfo.tyData.sBoardId	:= tyXMLTableNxt.sValue;
		END_IF

	ELSIF (tyXMLTableCurr.sTitle = 'AT') AND (sCurrValueLowerCase = 'boardidcreatedby') THEN

		p_tySendBoardInfo.tyAvl.bBoardIdCreatedBy	:= TRUE;

		IF tyXMLTableNxt.sTitle = 'AV' THEN
			p_tySendBoardInfo.tyData.sBoardIdCreatedBy	:= tyXMLTableNxt.sValue;
		END_IF

	ELSIF (tyXMLTableCurr.sTitle = 'AT') AND (sCurrValueLowerCase = 'failedboard') THEN

		p_tySendBoardInfo.tyAvl.bFailedBoard	:= TRUE;

		IF tyXMLTableNxt.sTitle = 'AV' THEN
			IF tyXMLTableNxt.sValue = '1' THEN
				p_tySendBoardInfo.tyData.eFailedBoard	:= HermesGoodBoard;
			ELSIF tyXMLTableNxt.sValue = '2' THEN
				p_tySendBoardInfo.tyData.eFailedBoard	:= HermesFailedBoard;
			ELSE
				p_tySendBoardInfo.tyData.eFailedBoard	:= HermesUnknownBoard;
			END_IF
		END_IF

	ELSIF (tyXMLTableCurr.sTitle = 'AT') AND (sCurrValueLowerCase = 'producttypeid') THEN

		p_tySendBoardInfo.tyAvl.bProductTypeId	:= TRUE;

		IF tyXMLTableNxt.sTitle = 'AV' THEN
			p_tySendBoardInfo.tyData.sProductTypeId	:= tyXMLTableNxt.sValue;
		END_IF

	ELSIF (tyXMLTableCurr.sTitle = 'AT') AND (sCurrValueLowerCase = 'flippedboard') THEN

		p_tySendBoardInfo.tyAvl.bFlippedBoard	:= TRUE;

		IF tyXMLTableNxt.sTitle = 'AV' THEN
			IF tyXMLTableNxt.sValue = '1' THEN
				p_tySendBoardInfo.tyData.eFlippedBoard	:= HermesFlippedBoardTopSideUp;
			ELSIF tyXMLTableNxt.sValue = '2' THEN
				p_tySendBoardInfo.tyData.eFlippedBoard	:= HermesFlippedBoardBtmSideUp;
			ELSE
				p_tySendBoardInfo.tyData.eFlippedBoard	:= HermesFlippedBoardUnknownSide;
			END_IF
		END_IF

	ELSIF (tyXMLTableCurr.sTitle = 'AT') AND (sCurrValueLowerCase = 'topbarcode') THEN

		p_tySendBoardInfo.tyAvl.bTopBarcode	:= TRUE;

		IF tyXMLTableNxt.sTitle = 'AV' THEN
			p_tySendBoardInfo.tyData.sTopBarcode	:= tyXMLTableNxt.sValue;
		END_IF

	ELSIF (tyXMLTableCurr.sTitle = 'AT') AND (sCurrValueLowerCase = 'bottombarcode') THEN

		p_tySendBoardInfo.tyAvl.bBottomBarcode	:= TRUE;

		IF tyXMLTableNxt.sTitle = 'AV' THEN
			p_tySendBoardInfo.tyData.sBottomBarcode	:= tyXMLTableNxt.sValue;
		END_IF

	ELSIF (tyXMLTableCurr.sTitle = 'AT') AND (sCurrValueLowerCase = 'length') THEN

		p_tySendBoardInfo.tyAvl.bLength	:= TRUE;

		IF tyXMLTableNxt.sTitle = 'AV' THEN
			p_tySendBoardInfo.tyData.rLength	:= STRING_TO_REAL(tyXMLTableNxt.sValue);
		END_IF

	ELSIF (tyXMLTableCurr.sTitle = 'AT') AND (sCurrValueLowerCase = 'width') THEN

		p_tySendBoardInfo.tyAvl.bWidth	:= TRUE;

		IF tyXMLTableNxt.sTitle = 'AV' THEN
			p_tySendBoardInfo.tyData.rWidth	:= STRING_TO_REAL(tyXMLTableNxt.sValue);
		END_IF

	ELSIF (tyXMLTableCurr.sTitle = 'AT') AND (sCurrValueLowerCase = 'thickness') THEN

		p_tySendBoardInfo.tyAvl.bThickness	:= TRUE;

		IF tyXMLTableNxt.sTitle = 'AV' THEN
			p_tySendBoardInfo.tyData.rThickness	:= STRING_TO_REAL(tyXMLTableNxt.sValue);
		END_IF

	ELSIF (tyXMLTableCurr.sTitle = 'AT') AND (sCurrValueLowerCase = 'topclearanceheight') THEN

		p_tySendBoardInfo.tyAvl.bTopClearanceHeight	:= TRUE;

		IF tyXMLTableNxt.sTitle = 'AV' THEN
			p_tySendBoardInfo.tyData.rTopClearanceHeight	:= STRING_TO_REAL(tyXMLTableNxt.sValue);
		END_IF

	ELSIF (tyXMLTableCurr.sTitle = 'AT') AND (sCurrValueLowerCase = 'bottomclearanceheight') THEN

		p_tySendBoardInfo.tyAvl.bBottomClearanceHeight	:= TRUE;

		IF tyXMLTableNxt.sTitle = 'AV' THEN
			p_tySendBoardInfo.tyData.rBottomClearanceHeight	:= STRING_TO_REAL(tyXMLTableNxt.sValue);
		END_IF

	ELSIF (tyXMLTableCurr.sTitle = 'AT') AND (sCurrValueLowerCase = 'weight') THEN

		p_tySendBoardInfo.tyAvl.bWeight	:= TRUE;

		IF tyXMLTableNxt.sTitle = 'AV' THEN
			p_tySendBoardInfo.tyData.rWeight	:= STRING_TO_REAL(tyXMLTableNxt.sValue);
		END_IF

	ELSIF (tyXMLTableCurr.sTitle = 'AT') AND (sCurrValueLowerCase = 'workorderid') THEN

		p_tySendBoardInfo.tyAvl.bWorkOrderId	:= TRUE;

		IF tyXMLTableNxt.sTitle = 'AV' THEN
			p_tySendBoardInfo.tyData.sWorkOrderId	:= tyXMLTableNxt.sValue;
		END_IF

	ELSIF (tyXMLTableCurr.sTitle = 'AT') AND (sCurrValueLowerCase = 'batchid') THEN

		p_tySendBoardInfo.tyAvl.bBatchId	:= TRUE;

		IF tyXMLTableNxt.sTitle = 'AV' THEN
			p_tySendBoardInfo.tyData.sBatchId	:= tyXMLTableNxt.sValue;
		END_IF

	END_IF

END_FUNCTION
```

#### fHermesParseBoardArrived.st
```iecst
(* Hermes Parse XML Table Data For Board Arrived*)
FUNCTION fHermesParseBoardArrived

	fHermesParseBoardArrived	:= TRUE;

	IF (tyXMLTableCurr.sTitle = 'AT') AND (sCurrValueLowerCase = 'machineid') THEN

		p_tyBoardArrived.tyAvl.bMachineId	:= TRUE;

		IF tyXMLTableNxt.sTitle = 'AV' THEN
			p_tyBoardArrived.tyData.sMachineId	:= tyXMLTableNxt.sValue;
		END_IF

	ELSIF (tyXMLTableCurr.sTitle = 'AT') AND (sCurrValueLowerCase = 'upstreamlaneid') THEN

		p_tyBoardArrived.tyAvl.bUpstreamLaneId	:= TRUE;

		IF tyXMLTableNxt.sTitle = 'AV' THEN
			p_tyBoardArrived.tyData.iUpstreamLaneId	:= STRING_TO_INT(tyXMLTableNxt.sValue);
		END_IF

	ELSIF (tyXMLTableCurr.sTitle = 'AT') AND (sCurrValueLowerCase = 'upstreaminterfaceid') THEN

		p_tyBoardArrived.tyAvl.bUpstreamInterfaceId	:= TRUE;

		IF tyXMLTableNxt.sTitle = 'AV' THEN
			p_tyBoardArrived.tyData.sUpstreamInterfaceId	:= tyXMLTableNxt.sValue;
		END_IF

	ELSIF (tyXMLTableCurr.sTitle = 'AT') AND (sCurrValueLowerCase = 'magazineid') THEN

		p_tyBoardArrived.tyAvl.bMagazineId	:= TRUE;

		IF tyXMLTableNxt.sTitle = 'AV' THEN
			p_tyBoardArrived.tyData.sMagazineId	:= tyXMLTableNxt.sValue;
		END_IF

	ELSIF (tyXMLTableCurr.sTitle = 'AT') AND (sCurrValueLowerCase = 'slotid') THEN

		p_tyBoardArrived.tyAvl.bSlotId	:= TRUE;

		IF tyXMLTableNxt.sTitle = 'AV' THEN
			p_tyBoardArrived.tyData.iSlotId	:= STRING_TO_INT(tyXMLTableNxt.sValue);
		END_IF

	ELSIF (tyXMLTableCurr.sTitle = 'AT') AND (sCurrValueLowerCase = 'boardtransfer') THEN

		p_tyBoardArrived.tyAvl.bBoardTransfer	:= TRUE;

		IF tyXMLTableNxt.sTitle = 'AV' THEN
			IF tyXMLTableNxt.sValue = '1' THEN
				p_tyBoardArrived.tyData.eBoadTransfer	:= HermesTransferred;
			ELSIF tyXMLTableNxt.sValue = '2' THEN
				p_tyBoardArrived.tyData.eBoadTransfer	:= HermesLoaded;
			ELSIF tyXMLTableNxt.sValue = '3' THEN
				p_tyBoardArrived.tyData.eBoadTransfer	:= HermesInserted;
			END_IF
		END_IF

	ELSIF (tyXMLTableCurr.sTitle = 'AT') AND (sCurrValueLowerCase = 'boardid') THEN

		p_tyBoardArrived.tyAvl.bBoardId	:= TRUE;

		IF tyXMLTableNxt.sTitle = 'AV' THEN
			p_tyBoardArrived.tyData.sBoardId	:= tyXMLTableNxt.sValue;
		END_IF

	ELSIF (tyXMLTableCurr.sTitle = 'AT') AND (sCurrValueLowerCase = 'boardidcreatedby') THEN

		p_tyBoardArrived.tyAvl.bBoardIdCreatedBy	:= TRUE;

		IF tyXMLTableNxt.sTitle = 'AV' THEN
			p_tyBoardArrived.tyData.sBoardIdCreatedBy	:= tyXMLTableNxt.sValue;
		END_IF

	ELSIF (tyXMLTableCurr.sTitle = 'AT') AND (sCurrValueLowerCase = 'failedboard') THEN

		p_tyBoardArrived.tyAvl.bFailedBoard	:= TRUE;

		IF tyXMLTableNxt.sTitle = 'AV' THEN
			IF tyXMLTableNxt.sValue = '1' THEN
				p_tyBoardArrived.tyData.eFailedBoard	:= HermesGoodBoard;
			ELSIF tyXMLTableNxt.sValue = '2' THEN
				p_tyBoardArrived.tyData.eFailedBoard	:= HermesFailedBoard;
			ELSE
				p_tyBoardArrived.tyData.eFailedBoard	:= HermesUnknownBoard;
			END_IF
		END_IF

	ELSIF (tyXMLTableCurr.sTitle = 'AT') AND (sCurrValueLowerCase = 'producttypeid') THEN

		p_tyBoardArrived.tyAvl.bProductTypeId	:= TRUE;

		IF tyXMLTableNxt.sTitle = 'AV' THEN
			p_tyBoardArrived.tyData.sProductTypeId	:= tyXMLTableNxt.sValue;
		END_IF

	ELSIF (tyXMLTableCurr.sTitle = 'AT') AND (sCurrValueLowerCase = 'flippedboard') THEN

		p_tyBoardArrived.tyAvl.bFlippedBoard	:= TRUE;

		IF tyXMLTableNxt.sTitle = 'AV' THEN
			IF tyXMLTableNxt.sValue = '1' THEN
				p_tyBoardArrived.tyData.eFlippedBoard	:= HermesFlippedBoardTopSideUp;
			ELSIF tyXMLTableNxt.sValue = '2' THEN
				p_tyBoardArrived.tyData.eFlippedBoard	:= HermesFlippedBoardBtmSideUp;
			ELSE
				p_tyBoardArrived.tyData.eFlippedBoard	:= HermesFlippedBoardUnknownSide;
			END_IF
		END_IF

	ELSIF (tyXMLTableCurr.sTitle = 'AT') AND (sCurrValueLowerCase = 'topbarcode') THEN

		p_tyBoardArrived.tyAvl.bTopBarcode	:= TRUE;

		IF tyXMLTableNxt.sTitle = 'AV' THEN
			p_tyBoardArrived.tyData.sTopBarcode	:= tyXMLTableNxt.sValue;
		END_IF

	ELSIF (tyXMLTableCurr.sTitle = 'AT') AND (sCurrValueLowerCase = 'bottombarcode') THEN

		p_tyBoardArrived.tyAvl.bBottomBarcode	:= TRUE;

		IF tyXMLTableNxt.sTitle = 'AV' THEN
			p_tyBoardArrived.tyData.sBottomBarcode	:= tyXMLTableNxt.sValue;
		END_IF

	ELSIF (tyXMLTableCurr.sTitle = 'AT') AND (sCurrValueLowerCase = 'length') THEN

		p_tyBoardArrived.tyAvl.bLength	:= TRUE;

		IF tyXMLTableNxt.sTitle = 'AV' THEN
			p_tyBoardArrived.tyData.rLength	:= STRING_TO_REAL(tyXMLTableNxt.sValue);
		END_IF

	ELSIF (tyXMLTableCurr.sTitle = 'AT') AND (sCurrValueLowerCase = 'width') THEN

		p_tyBoardArrived.tyAvl.bWidth	:= TRUE;

		IF tyXMLTableNxt.sTitle = 'AV' THEN
			p_tyBoardArrived.tyData.rWidth	:= STRING_TO_REAL(tyXMLTableNxt.sValue);
		END_IF

	ELSIF (tyXMLTableCurr.sTitle = 'AT') AND (sCurrValueLowerCase = 'thickness') THEN

		p_tyBoardArrived.tyAvl.bThickness	:= TRUE;

		IF tyXMLTableNxt.sTitle = 'AV' THEN
			p_tyBoardArrived.tyData.rThickness	:= STRING_TO_REAL(tyXMLTableNxt.sValue);
		END_IF

	ELSIF (tyXMLTableCurr.sTitle = 'AT') AND (sCurrValueLowerCase = 'conveyorspeed') THEN

		p_tyBoardArrived.tyAvl.bConveyorSpeed	:= TRUE;

		IF tyXMLTableNxt.sTitle = 'AV' THEN
			p_tyBoardArrived.tyData.rConveyorSpeed	:= STRING_TO_REAL(tyXMLTableNxt.sValue);
		END_IF

	ELSIF (tyXMLTableCurr.sTitle = 'AT') AND (sCurrValueLowerCase = 'topclearanceheight') THEN

		p_tyBoardArrived.tyAvl.bTopClearanceHeight	:= TRUE;

		IF tyXMLTableNxt.sTitle = 'AV' THEN
			p_tyBoardArrived.tyData.rTopClearanceHeight	:= STRING_TO_REAL(tyXMLTableNxt.sValue);
		END_IF

	ELSIF (tyXMLTableCurr.sTitle = 'AT') AND (sCurrValueLowerCase = 'bottomclearanceheight') THEN

		p_tyBoardArrived.tyAvl.bBottomClearanceHeight	:= TRUE;

		IF tyXMLTableNxt.sTitle = 'AV' THEN
			p_tyBoardArrived.tyData.rBottomClearanceHeight	:= STRING_TO_REAL(tyXMLTableNxt.sValue);
		END_IF

	ELSIF (tyXMLTableCurr.sTitle = 'AT') AND (sCurrValueLowerCase = 'weight') THEN

		p_tyBoardArrived.tyAvl.bWeight	:= TRUE;

		IF tyXMLTableNxt.sTitle = 'AV' THEN
			p_tyBoardArrived.tyData.rWeight	:= STRING_TO_REAL(tyXMLTableNxt.sValue);
		END_IF

	ELSIF (tyXMLTableCurr.sTitle = 'AT') AND (sCurrValueLowerCase = 'workorderid') THEN

		p_tyBoardArrived.tyAvl.bWorkOrderId	:= TRUE;

		IF tyXMLTableNxt.sTitle = 'AV' THEN
			p_tyBoardArrived.tyData.sWorkOrdedId	:= tyXMLTableNxt.sValue;
		END_IF

	ELSIF (tyXMLTableCurr.sTitle = 'AT') AND (sCurrValueLowerCase = 'batchid') THEN

		p_tyBoardArrived.tyAvl.bBatchId	:= TRUE;

		IF tyXMLTableNxt.sTitle = 'AV' THEN
			p_tyBoardArrived.tyData.sBatchId	:= tyXMLTableNxt.sValue;
		END_IF

	ELSIF (tyXMLTableCurr.sTitle = 'AT') AND (sCurrValueLowerCase = 'route') THEN

		p_tyBoardArrived.tyAvl.bRoute	:= TRUE;

		IF tyXMLTableNxt.sTitle = 'AV' THEN
			p_tyBoardArrived.tyData.iRoute	:= STRING_TO_INT(tyXMLTableNxt.sValue);
		END_IF
	ELSIF (tyXMLTableCurr.sTitle = 'AT') AND (sCurrValueLowerCase = 'action') THEN

		p_tyBoardArrived.tyAvl.bAction	:= TRUE;

		IF tyXMLTableNxt.sTitle = 'AV' THEN
			p_tyBoardArrived.tyData.iAction	:= STRING_TO_INT(tyXMLTableNxt.sValue);
		END_IF
	END_IF

END_FUNCTION
```

#### fHermesParseBoardDeparted.st
```iecst
(* Hermes Parse XML Table Data For Board Departed*)
FUNCTION fHermesParseBoardDeparted

	fHermesParseBoardDeparted	:= TRUE;

	IF (tyXMLTableCurr.sTitle = 'AT') AND (sCurrValueLowerCase = 'machineid') THEN

		p_tyBoardDeparted.tyAvl.bMachineId	:= TRUE;

		IF tyXMLTableNxt.sTitle = 'AV' THEN
			p_tyBoardDeparted.tyData.sMachineId	:= tyXMLTableNxt.sValue;
		END_IF

	ELSIF (tyXMLTableCurr.sTitle = 'AT') AND (sCurrValueLowerCase = 'downstreamlaneid') THEN

		p_tyBoardDeparted.tyAvl.bDownstreamLaneId	:= TRUE;

		IF tyXMLTableNxt.sTitle = 'AV' THEN
			p_tyBoardDeparted.tyData.iDownstreamLaneId	:= STRING_TO_INT(tyXMLTableNxt.sValue);
		END_IF

	ELSIF (tyXMLTableCurr.sTitle = 'AT') AND (sCurrValueLowerCase = 'downstreaminterfaceid') THEN

		p_tyBoardDeparted.tyAvl.bDownstreamInterfaceId	:= TRUE;

		IF tyXMLTableNxt.sTitle = 'AV' THEN
			p_tyBoardDeparted.tyData.sDownstreamInterfaceId	:= tyXMLTableNxt.sValue;
		END_IF

	ELSIF (tyXMLTableCurr.sTitle = 'AT') AND (sCurrValueLowerCase = 'magazineid') THEN

		p_tyBoardDeparted.tyAvl.bMagazineId	:= TRUE;

		IF tyXMLTableNxt.sTitle = 'AV' THEN
			p_tyBoardDeparted.tyData.sMagazineId	:= tyXMLTableNxt.sValue;
		END_IF

	ELSIF (tyXMLTableCurr.sTitle = 'AT') AND (sCurrValueLowerCase = 'slotid') THEN

		p_tyBoardDeparted.tyAvl.bSlotId	:= TRUE;

		IF tyXMLTableNxt.sTitle = 'AV' THEN
			p_tyBoardDeparted.tyData.iSlotId	:= STRING_TO_INT(tyXMLTableNxt.sValue);
		END_IF

	ELSIF (tyXMLTableCurr.sTitle = 'AT') AND (sCurrValueLowerCase = 'boardtransfer') THEN

		p_tyBoardDeparted.tyAvl.bBoardTransfer	:= TRUE;

		IF tyXMLTableNxt.sTitle = 'AV' THEN
			IF tyXMLTableNxt.sValue = '1' THEN
				p_tyBoardDeparted.tyData.eBoadTransfer	:= HermesTransferred;
			ELSIF tyXMLTableNxt.sValue = '2' THEN
				p_tyBoardDeparted.tyData.eBoadTransfer	:= HermesLoaded;
			ELSIF tyXMLTableNxt.sValue = '3' THEN
				p_tyBoardDeparted.tyData.eBoadTransfer	:= HermesInserted;
			END_IF
		END_IF

	ELSIF (tyXMLTableCurr.sTitle = 'AT') AND (sCurrValueLowerCase = 'boardid') THEN

		p_tyBoardDeparted.tyAvl.bBoardId	:= TRUE;

		IF tyXMLTableNxt.sTitle = 'AV' THEN
			p_tyBoardDeparted.tyData.sBoardId	:= tyXMLTableNxt.sValue;
		END_IF

	ELSIF (tyXMLTableCurr.sTitle = 'AT') AND (sCurrValueLowerCase = 'boardidcreatedby') THEN

		p_tyBoardDeparted.tyAvl.bBoardIdCreatedBy	:= TRUE;

		IF tyXMLTableNxt.sTitle = 'AV' THEN
			p_tyBoardDeparted.tyData.sBoardIdCreatedBy	:= tyXMLTableNxt.sValue;
		END_IF

	ELSIF (tyXMLTableCurr.sTitle = 'AT') AND (sCurrValueLowerCase = 'failedboard') THEN

		p_tyBoardDeparted.tyAvl.bFailedBoard	:= TRUE;

		IF tyXMLTableNxt.sTitle = 'AV' THEN
			IF tyXMLTableNxt.sValue = '1' THEN
				p_tyBoardDeparted.tyData.eFailedBoard	:= HermesGoodBoard;
			ELSIF tyXMLTableNxt.sValue = '2' THEN
				p_tyBoardDeparted.tyData.eFailedBoard	:= HermesFailedBoard;
			ELSE
				p_tyBoardDeparted.tyData.eFailedBoard	:= HermesUnknownBoard;
			END_IF
		END_IF

	ELSIF (tyXMLTableCurr.sTitle = 'AT') AND (sCurrValueLowerCase = 'producttypeid') THEN

		p_tyBoardDeparted.tyAvl.bProductTypeId	:= TRUE;

		IF tyXMLTableNxt.sTitle = 'AV' THEN
			p_tyBoardDeparted.tyData.sProductTypeId	:= tyXMLTableNxt.sValue;
		END_IF

	ELSIF (tyXMLTableCurr.sTitle = 'AT') AND (sCurrValueLowerCase = 'flippedboard') THEN

		p_tyBoardDeparted.tyAvl.bFlippedBoard	:= TRUE;

		IF tyXMLTableNxt.sTitle = 'AV' THEN
			IF tyXMLTableNxt.sValue = '1' THEN
				p_tyBoardDeparted.tyData.eFlippedBoard	:= HermesFlippedBoardTopSideUp;
			ELSIF tyXMLTableNxt.sValue = '2' THEN
				p_tyBoardDeparted.tyData.eFlippedBoard	:= HermesFlippedBoardBtmSideUp;
			ELSE
				p_tyBoardDeparted.tyData.eFlippedBoard	:= HermesFlippedBoardUnknownSide;
			END_IF
		END_IF

	ELSIF (tyXMLTableCurr.sTitle = 'AT') AND (sCurrValueLowerCase = 'topbarcode') THEN

		p_tyBoardDeparted.tyAvl.bTopBarcode	:= TRUE;

		IF tyXMLTableNxt.sTitle = 'AV' THEN
			p_tyBoardDeparted.tyData.sTopBarcode	:= tyXMLTableNxt.sValue;
		END_IF

	ELSIF (tyXMLTableCurr.sTitle = 'AT') AND (sCurrValueLowerCase = 'bottombarcode') THEN

		p_tyBoardDeparted.tyAvl.bBottomBarcode	:= TRUE;

		IF tyXMLTableNxt.sTitle = 'AV' THEN
			p_tyBoardDeparted.tyData.sBottomBarcode	:= tyXMLTableNxt.sValue;
		END_IF

	ELSIF (tyXMLTableCurr.sTitle = 'AT') AND (sCurrValueLowerCase = 'length') THEN

		p_tyBoardDeparted.tyAvl.bLength	:= TRUE;

		IF tyXMLTableNxt.sTitle = 'AV' THEN
			p_tyBoardDeparted.tyData.rLength	:= STRING_TO_REAL(tyXMLTableNxt.sValue);
		END_IF

	ELSIF (tyXMLTableCurr.sTitle = 'AT') AND (sCurrValueLowerCase = 'width') THEN

		p_tyBoardDeparted.tyAvl.bWidth	:= TRUE;

		IF tyXMLTableNxt.sTitle = 'AV' THEN
			p_tyBoardDeparted.tyData.rWidth	:= STRING_TO_REAL(tyXMLTableNxt.sValue);
		END_IF

	ELSIF (tyXMLTableCurr.sTitle = 'AT') AND (sCurrValueLowerCase = 'thickness') THEN

		p_tyBoardDeparted.tyAvl.bThickness	:= TRUE;

		IF tyXMLTableNxt.sTitle = 'AV' THEN
			p_tyBoardDeparted.tyData.rThickness	:= STRING_TO_REAL(tyXMLTableNxt.sValue);
		END_IF

	ELSIF (tyXMLTableCurr.sTitle = 'AT') AND (sCurrValueLowerCase = 'conveyorspeed') THEN

		p_tyBoardDeparted.tyAvl.bConveyorSpeed	:= TRUE;

		IF tyXMLTableNxt.sTitle = 'AV' THEN
			p_tyBoardDeparted.tyData.rConveyorSpeed	:= STRING_TO_REAL(tyXMLTableNxt.sValue);
		END_IF

	ELSIF (tyXMLTableCurr.sTitle = 'AT') AND (sCurrValueLowerCase = 'topclearanceheight') THEN

		p_tyBoardDeparted.tyAvl.bTopClearanceHeight	:= TRUE;

		IF tyXMLTableNxt.sTitle = 'AV' THEN
			p_tyBoardDeparted.tyData.rTopClearanceHeight	:= STRING_TO_REAL(tyXMLTableNxt.sValue);
		END_IF

	ELSIF (tyXMLTableCurr.sTitle = 'AT') AND (sCurrValueLowerCase = 'bottomclearanceheight') THEN

		p_tyBoardDeparted.tyAvl.bBottomClearanceHeight	:= TRUE;

		IF tyXMLTableNxt.sTitle = 'AV' THEN
			p_tyBoardDeparted.tyData.rBottomClearanceHeight	:= STRING_TO_REAL(tyXMLTableNxt.sValue);
		END_IF

	ELSIF (tyXMLTableCurr.sTitle = 'AT') AND (sCurrValueLowerCase = 'weight') THEN

		p_tyBoardDeparted.tyAvl.bWeight	:= TRUE;

		IF tyXMLTableNxt.sTitle = 'AV' THEN
			p_tyBoardDeparted.tyData.rWeight	:= STRING_TO_REAL(tyXMLTableNxt.sValue);
		END_IF

	ELSIF (tyXMLTableCurr.sTitle = 'AT') AND (sCurrValueLowerCase = 'workorderid') THEN

		p_tyBoardDeparted.tyAvl.bWorkOrderId	:= TRUE;

		IF tyXMLTableNxt.sTitle = 'AV' THEN
			p_tyBoardDeparted.tyData.sWorkOrdedId	:= tyXMLTableNxt.sValue;
		END_IF

	ELSIF (tyXMLTableCurr.sTitle = 'AT') AND (sCurrValueLowerCase = 'batchid') THEN

		p_tyBoardDeparted.tyAvl.bBatchId	:= TRUE;

		IF tyXMLTableNxt.sTitle = 'AV' THEN
			p_tyBoardDeparted.tyData.sBatchId	:= tyXMLTableNxt.sValue;
		END_IF
	ELSIF (tyXMLTableCurr.sTitle = 'AT') AND (sCurrValueLowerCase = 'route') THEN

		p_tyBoardDeparted.tyAvl.bRoute	:= TRUE;

		IF tyXMLTableNxt.sTitle = 'AV' THEN
			p_tyBoardDeparted.tyData.iRoute	:= STRING_TO_INT(tyXMLTableNxt.sValue);
		END_IF
	ELSIF (tyXMLTableCurr.sTitle = 'AT') AND (sCurrValueLowerCase = 'action') THEN

		p_tyBoardDeparted.tyAvl.bAction	:= TRUE;

		IF tyXMLTableNxt.sTitle = 'AV' THEN
			p_tyBoardDeparted.tyData.iAction	:= STRING_TO_INT(tyXMLTableNxt.sValue);
		END_IF
	END_IF

END_FUNCTION
```

#### fHermesParseQueryWorkOrderInfo.st
```iecst
(* Hermes Parse XML Table Data For Query Board Info *)
FUNCTION fHermesParseQueryWorkOrderInfo

	fHermesParseQueryWorkOrderInfo	:= TRUE;

	IF (tyXMLTableCurr.sTitle = 'AT') AND (sCurrValueLowerCase = 'queryid') THEN

		p_tyQueryWorkOrderInfo.tyAvl.bQueryId	:= TRUE;

		IF tyXMLTableNxt.sTitle = 'AV' THEN
			p_tyQueryWorkOrderInfo.tyData.sQueryId	:= tyXMLTableNxt.sValue;
		END_IF

	ELSIF (tyXMLTableCurr.sTitle = 'AT') AND (sCurrValueLowerCase = 'machineid') THEN

		p_tyQueryWorkOrderInfo.tyAvl.bMachineId   := TRUE;

		IF tyXMLTableNxt.sTitle = 'AV' THEN
			p_tyQueryWorkOrderInfo.tyData.sMachineId	:= tyXMLTableNxt.sValue;
		END_IF

	ELSIF (tyXMLTableCurr.sTitle = 'AT') AND (sCurrValueLowerCase = 'magazineid') THEN

		p_tyQueryWorkOrderInfo.tyAvl.bMagazineId   := TRUE;

		IF tyXMLTableNxt.sTitle = 'AV' THEN
			p_tyQueryWorkOrderInfo.tyData.sMagazineId	:= tyXMLTableNxt.sValue;
		END_IF

	ELSIF (tyXMLTableCurr.sTitle = 'AT') AND (sCurrValueLowerCase = 'slotid') THEN

		p_tyQueryWorkOrderInfo.tyAvl.bSlotId   := TRUE;

		IF tyXMLTableNxt.sTitle = 'AV' THEN
			p_tyQueryWorkOrderInfo.tyData.iSlotId	:= STRING_TO_INT(tyXMLTableNxt.sValue);
		END_IF

	ELSIF (tyXMLTableCurr.sTitle = 'AT') AND (sCurrValueLowerCase = 'barcode') THEN

		p_tyQueryWorkOrderInfo.tyAvl.bBarcode   := TRUE;

		IF tyXMLTableNxt.sTitle = 'AV' THEN
			p_tyQueryWorkOrderInfo.tyData.sBarcode	:= tyXMLTableNxt.sValue;
		END_IF

	END_IF

END_FUNCTION
```

#### fHermesParseSendWorkOrderInfo.st
```iecst
(* Hermes Parse XML Table Data For Send Work Order Info*)
FUNCTION fHermesParseSendWorkOrderInfo

	fHermesParseSendWorkOrderInfo	:= TRUE;

	IF (tyXMLTableCurr.sTitle = 'AT') AND (sCurrValueLowerCase = 'queryid') THEN

	    p_tySendWorkOrderInfo.tyAvl.bQueryId	:= TRUE;

     	IF tyXMLTableNxt.sTitle = 'AV' THEN
		p_tySendWorkOrderInfo.tyData.sQueryId	:= tyXMLTableNxt.sValue;
    	END_IF

	ELSIF (tyXMLTableCurr.sTitle = 'AT') AND (sCurrValueLowerCase = 'workorderid') THEN

	    p_tySendWorkOrderInfo.tyAvl.bWorkOrderId	:= TRUE;

    	IF tyXMLTableNxt.sTitle = 'AV' THEN
		p_tySendWorkOrderInfo.tyData.sWorkOrderId	:= tyXMLTableNxt.sValue;
		END_IF

	ELSIF (tyXMLTableCurr.sTitle = 'AT') AND (sCurrValueLowerCase = 'batchid') THEN

		p_tySendWorkOrderInfo.tyAvl.bBatchId	:= TRUE;

		IF tyXMLTableNxt.sTitle = 'AV' THEN
			p_tySendWorkOrderInfo.tyData.sBatchId	:= tyXMLTableNxt.sValue;
		END_IF

	ELSIF (tyXMLTableCurr.sTitle = 'AT') AND (sCurrValueLowerCase = 'boardid') THEN

		p_tySendWorkOrderInfo.tyAvl.bBoardId	:= TRUE;

		IF tyXMLTableNxt.sTitle = 'AV' THEN
			p_tySendWorkOrderInfo.tyData.sBoardId	:= tyXMLTableNxt.sValue;
		END_IF

	ELSIF (tyXMLTableCurr.sTitle = 'AT') AND (sCurrValueLowerCase = 'boardidcreatedby') THEN

		p_tySendWorkOrderInfo.tyAvl.bBoardIdCreatedBy	:= TRUE;

		IF tyXMLTableNxt.sTitle = 'AV' THEN
			p_tySendWorkOrderInfo.tyData.sBoardIdCreatedBy	:= tyXMLTableNxt.sValue;
		END_IF

	ELSIF (tyXMLTableCurr.sTitle = 'AT') AND (sCurrValueLowerCase = 'failedboard') THEN

		p_tySendWorkOrderInfo.tyAvl.bFailedBoard	:= TRUE;

		IF tyXMLTableNxt.sTitle = 'AV' THEN
			IF tyXMLTableNxt.sValue = '1' THEN
				p_tySendWorkOrderInfo.tyData.eFailedBoard	:= HermesGoodBoard;
			ELSIF tyXMLTableNxt.sValue = '2' THEN
				p_tySendWorkOrderInfo.tyData.eFailedBoard	:= HermesFailedBoard;
			ELSE
				p_tySendWorkOrderInfo.tyData.eFailedBoard	:= HermesUnknownBoard;
			END_IF
		END_IF

	ELSIF (tyXMLTableCurr.sTitle = 'AT') AND (sCurrValueLowerCase = 'producttypeid') THEN

		p_tySendWorkOrderInfo.tyAvl.bProductTypeId	:= TRUE;

		IF tyXMLTableNxt.sTitle = 'AV' THEN
			p_tySendWorkOrderInfo.tyData.sProductTypeId	:= tyXMLTableNxt.sValue;
		END_IF

	ELSIF (tyXMLTableCurr.sTitle = 'AT') AND (sCurrValueLowerCase = 'flippedboard') THEN

		p_tySendWorkOrderInfo.tyAvl.bFlippedBoard	:= TRUE;

		IF tyXMLTableNxt.sTitle = 'AV' THEN
			IF tyXMLTableNxt.sValue = '1' THEN
				p_tySendWorkOrderInfo.tyData.eFlippedBoard	:= HermesFlippedBoardTopSideUp;
			ELSIF tyXMLTableNxt.sValue = '2' THEN
				p_tySendWorkOrderInfo.tyData.eFlippedBoard	:= HermesFlippedBoardBtmSideUp;
			ELSE
				p_tySendWorkOrderInfo.tyData.eFlippedBoard	:= HermesFlippedBoardUnknownSide;
			END_IF
		END_IF

	ELSIF (tyXMLTableCurr.sTitle = 'AT') AND (sCurrValueLowerCase = 'topbarcode') THEN

		p_tySendWorkOrderInfo.tyAvl.bTopBarcode	:= TRUE;

		IF tyXMLTableNxt.sTitle = 'AV' THEN
			p_tySendWorkOrderInfo.tyData.sTopBarcode	:= tyXMLTableNxt.sValue;
		END_IF

	ELSIF (tyXMLTableCurr.sTitle = 'AT') AND (sCurrValueLowerCase = 'bottombarcode') THEN

		p_tySendWorkOrderInfo.tyAvl.bBottomBarcode	:= TRUE;

		IF tyXMLTableNxt.sTitle = 'AV' THEN
			p_tySendWorkOrderInfo.tyData.sBottomBarcode	:= tyXMLTableNxt.sValue;
		END_IF

	ELSIF (tyXMLTableCurr.sTitle = 'AT') AND (sCurrValueLowerCase = 'length') THEN

		p_tySendWorkOrderInfo.tyAvl.bLength	:= TRUE;

		IF tyXMLTableNxt.sTitle = 'AV' THEN
			p_tySendWorkOrderInfo.tyData.rLength	:= STRING_TO_REAL(tyXMLTableNxt.sValue);
		END_IF

	ELSIF (tyXMLTableCurr.sTitle = 'AT') AND (sCurrValueLowerCase = 'width') THEN

		p_tySendWorkOrderInfo.tyAvl.bWidth	:= TRUE;

		IF tyXMLTableNxt.sTitle = 'AV' THEN
			p_tySendWorkOrderInfo.tyData.rWidth	:= STRING_TO_REAL(tyXMLTableNxt.sValue);
		END_IF

	ELSIF (tyXMLTableCurr.sTitle = 'AT') AND (sCurrValueLowerCase = 'thickness') THEN

		p_tySendWorkOrderInfo.tyAvl.bThickness	:= TRUE;

		IF tyXMLTableNxt.sTitle = 'AV' THEN
			p_tySendWorkOrderInfo.tyData.rThickness	:= STRING_TO_REAL(tyXMLTableNxt.sValue);
		END_IF

	ELSIF (tyXMLTableCurr.sTitle = 'AT') AND (sCurrValueLowerCase = 'conveyorspeed') THEN

		p_tySendWorkOrderInfo.tyAvl.bConveyorSpeed	:= TRUE;

		IF tyXMLTableNxt.sTitle = 'AV' THEN
			p_tySendWorkOrderInfo.tyData.rConveyorSpeed	:= STRING_TO_REAL(tyXMLTableNxt.sValue);
		END_IF

	ELSIF (tyXMLTableCurr.sTitle = 'AT') AND (sCurrValueLowerCase = 'topclearanceheight') THEN

		p_tySendWorkOrderInfo.tyAvl.bTopClearanceHeight	:= TRUE;

		IF tyXMLTableNxt.sTitle = 'AV' THEN
			p_tySendWorkOrderInfo.tyData.rTopClearanceHeight	:= STRING_TO_REAL(tyXMLTableNxt.sValue);
		END_IF

	ELSIF (tyXMLTableCurr.sTitle = 'AT') AND (sCurrValueLowerCase = 'bottomclearanceheight') THEN

		p_tySendWorkOrderInfo.tyAvl.bBottomClearanceHeight	:= TRUE;

		IF tyXMLTableNxt.sTitle = 'AV' THEN
			p_tySendWorkOrderInfo.tyData.rBottomClearanceHeight	:= STRING_TO_REAL(tyXMLTableNxt.sValue);
		END_IF

	ELSIF (tyXMLTableCurr.sTitle = 'AT') AND (sCurrValueLowerCase = 'weight') THEN

		p_tySendWorkOrderInfo.tyAvl.bWeight	:= TRUE;

		IF tyXMLTableNxt.sTitle = 'AV' THEN
			p_tySendWorkOrderInfo.tyData.rWeight	:= STRING_TO_REAL(tyXMLTableNxt.sValue);
		END_IF
	ELSIF (tyXMLTableCurr.sTitle = 'AT') AND (sCurrValueLowerCase = 'route') THEN

		p_tySendWorkOrderInfo.tyAvl.bRoute	:= TRUE;

		IF tyXMLTableNxt.sTitle = 'AV' THEN
			p_tySendWorkOrderInfo.tyData.iRoute	:= STRING_TO_INT(tyXMLTableNxt.sValue);
		END_IF

	END_IF

END_FUNCTION
```

#### fHermesParseCommand.st
```iecst
(* Hermes Parse XML Table Data For Send Work Order Info*)
FUNCTION fHermesParseCommand

	fHermesParseCommand	:= TRUE;

	IF (tyXMLTableCurr.sTitle = 'AT') AND (sCurrValueLowerCase = 'command') THEN

	    p_tyCommand.tyAvl.bCommand	:= TRUE;

		IF tyXMLTableNxt.sTitle = 'AV' THEN
			IF tyXMLTableNxt.sValue = '0' THEN
				p_tyCommand.tyData.eCommand	:= HermesCommandUndefined;
			ELSIF tyXMLTableNxt.sValue = '1' THEN
				p_tyCommand.tyData.eCommand	:= HermesCommandLockInputConveyor;
			ELSIF tyXMLTableNxt.sValue = '2' THEN
				p_tyCommand.tyData.eCommand	:= HermesCommandUnLockInputConveyor;
			ELSIF tyXMLTableNxt.sValue = '3' THEN
				p_tyCommand.tyData.eCommand	:= HermesCommandRequestPause;
			ELSIF tyXMLTableNxt.sValue = '4' THEN
				p_tyCommand.tyData.eCommand	:= HermesCommandConfirmPause;
			ELSIF tyXMLTableNxt.sValue = '5' THEN
				p_tyCommand.tyData.eCommand	:= HermesCommandResumeOperation;
			ELSIF tyXMLTableNxt.sValue = '1000' THEN
				p_tyCommand.tyData.eCommand	:= HermesCommandOvenInfeed;
			ELSIF tyXMLTableNxt.sValue = '1001' THEN
				p_tyCommand.tyData.eCommand	:= HermesCommandSelfDefine;
			END_IF
		END_IF

	END_IF

END_FUNCTION
```

#### fHermesFormCheckAlive.st
```iecst
(* Hermes Form Check Alive Table Data (Total Index Written In Table) *)
FUNCTION fHermesFormCheckAlive

	memset(ADR(pa_tyXMLTable) , 0 , SIZEOF(pa_tyXMLTable));
	iTotalIdxWrite	:= 0;

	fHermesGetTimestamp(ADR(sTimestamp) , tyDTStructure);

	pa_tyXMLTable[iTotalIdxWrite].sTitle	:= 'ST';
	pa_tyXMLTable[iTotalIdxWrite].sValue	:= 'Hermes';
	pa_tyXMLTable[iTotalIdxWrite].uiSize	:= LEN(pa_tyXMLTable[iTotalIdxWrite].sValue);

	iTotalIdxWrite	:= iTotalIdxWrite + 1;

	pa_tyXMLTable[iTotalIdxWrite].sTitle	:= 'AT';
	pa_tyXMLTable[iTotalIdxWrite].sValue	:= 'Timestamp';
	pa_tyXMLTable[iTotalIdxWrite].uiSize	:= LEN(pa_tyXMLTable[iTotalIdxWrite].sValue);

	iTotalIdxWrite	:= iTotalIdxWrite + 1;

	pa_tyXMLTable[iTotalIdxWrite].sTitle	:= 'AV';
	pa_tyXMLTable[iTotalIdxWrite].sValue	:= sTimestamp;
	pa_tyXMLTable[iTotalIdxWrite].uiSize	:= LEN(pa_tyXMLTable[iTotalIdxWrite].sValue);

	iTotalIdxWrite	:= iTotalIdxWrite + 1;

	pa_tyXMLTable[iTotalIdxWrite].sTitle	:= 'EN';
	pa_tyXMLTable[iTotalIdxWrite].sValue	:= '';
	pa_tyXMLTable[iTotalIdxWrite].uiSize	:= LEN(pa_tyXMLTable[iTotalIdxWrite].sValue);

	iTotalIdxWrite	:= iTotalIdxWrite + 1;

	pa_tyXMLTable[iTotalIdxWrite].sTitle	:= 'ST';
	pa_tyXMLTable[iTotalIdxWrite].sValue	:= 'CheckAlive';
	pa_tyXMLTable[iTotalIdxWrite].uiSize	:= LEN(pa_tyXMLTable[iTotalIdxWrite].sValue);

	iTotalIdxWrite	:= iTotalIdxWrite + 1;

	IF tyParameter.tyAvl.bType = TRUE THEN
		pa_tyXMLTable[iTotalIdxWrite].sTitle	:= 'AT';
		pa_tyXMLTable[iTotalIdxWrite].sValue	:= 'Type';
		pa_tyXMLTable[iTotalIdxWrite].uiSize	:= LEN(pa_tyXMLTable[iTotalIdxWrite].sValue);

		iTotalIdxWrite	:= iTotalIdxWrite + 1;

		pa_tyXMLTable[iTotalIdxWrite].sTitle	:= 'AV';
		pa_tyXMLTable[iTotalIdxWrite].sValue	:= DINT_TO_STRING(UDINT_TO_DINT(tyParameter.tyData.eType));
		pa_tyXMLTable[iTotalIdxWrite].uiSize	:= LEN(pa_tyXMLTable[iTotalIdxWrite].sValue);

		iTotalIdxWrite	:= iTotalIdxWrite + 1;
	END_IF

	IF tyParameter.tyAvl.bId = TRUE THEN
		pa_tyXMLTable[iTotalIdxWrite].sTitle	:= 'AT';
		pa_tyXMLTable[iTotalIdxWrite].sValue	:= 'Id';
		pa_tyXMLTable[iTotalIdxWrite].uiSize	:= LEN(pa_tyXMLTable[iTotalIdxWrite].sValue);

		iTotalIdxWrite	:= iTotalIdxWrite + 1;

		pa_tyXMLTable[iTotalIdxWrite].sTitle	:= 'AV';
		pa_tyXMLTable[iTotalIdxWrite].sValue	:= tyParameter.tyData.sId;
		pa_tyXMLTable[iTotalIdxWrite].uiSize	:= LEN(pa_tyXMLTable[iTotalIdxWrite].sValue);

		iTotalIdxWrite	:= iTotalIdxWrite + 1;
	END_IF

	pa_tyXMLTable[iTotalIdxWrite].sTitle	:= 'ES';
	pa_tyXMLTable[iTotalIdxWrite].sValue	:= '';
	pa_tyXMLTable[iTotalIdxWrite].uiSize	:= LEN(pa_tyXMLTable[iTotalIdxWrite].sValue);

	iTotalIdxWrite	:= iTotalIdxWrite + 1;

	pa_tyXMLTable[iTotalIdxWrite].sTitle	:= 'ET';
	pa_tyXMLTable[iTotalIdxWrite].sValue	:= 'Hermes';
	pa_tyXMLTable[iTotalIdxWrite].uiSize	:= LEN(pa_tyXMLTable[iTotalIdxWrite].sValue);

	iTotalIdxWrite	:= iTotalIdxWrite + 1;

	pa_tyXMLTable[iTotalIdxWrite].sTitle	:= 'EN';
	pa_tyXMLTable[iTotalIdxWrite].sValue	:= '';
	pa_tyXMLTable[iTotalIdxWrite].uiSize	:= LEN(pa_tyXMLTable[iTotalIdxWrite].sValue);

	iTotalIdxWrite	:= iTotalIdxWrite + 1;

	iTotalIdxWrite	:= fHermesFormCheckAlive;

END_FUNCTION
```

#### fHermesFormServiceDescription.st
```iecst
(* Hermes Form Service Description Table Data (Total Index Written In Table) *)
FUNCTION fHermesFormServiceDescription

	memset(ADR(pa_tyXMLTable) , 0 , SIZEOF(pa_tyXMLTable));
	iTotalIdxWrite	:= 0;

	fHermesGetTimestamp(ADR(sTimestamp) , tyDTStructure);

	pa_tyXMLTable[iTotalIdxWrite].sTitle	:= 'ST';
	pa_tyXMLTable[iTotalIdxWrite].sValue	:= 'Hermes';
	pa_tyXMLTable[iTotalIdxWrite].uiSize	:= LEN(pa_tyXMLTable[iTotalIdxWrite].sValue);

	iTotalIdxWrite	:= iTotalIdxWrite + 1;

	pa_tyXMLTable[iTotalIdxWrite].sTitle	:= 'AT';
	pa_tyXMLTable[iTotalIdxWrite].sValue	:= 'Timestamp';
	pa_tyXMLTable[iTotalIdxWrite].uiSize	:= LEN(pa_tyXMLTable[iTotalIdxWrite].sValue);

	iTotalIdxWrite	:= iTotalIdxWrite + 1;

	pa_tyXMLTable[iTotalIdxWrite].sTitle	:= 'AV';
	pa_tyXMLTable[iTotalIdxWrite].sValue	:= sTimestamp;
	pa_tyXMLTable[iTotalIdxWrite].uiSize	:= LEN(pa_tyXMLTable[iTotalIdxWrite].sValue);

	iTotalIdxWrite	:= iTotalIdxWrite + 1;

	pa_tyXMLTable[iTotalIdxWrite].sTitle	:= 'EN';
	pa_tyXMLTable[iTotalIdxWrite].sValue	:= '';
	pa_tyXMLTable[iTotalIdxWrite].uiSize	:= LEN(pa_tyXMLTable[iTotalIdxWrite].sValue);

	iTotalIdxWrite	:= iTotalIdxWrite + 1;

	pa_tyXMLTable[iTotalIdxWrite].sTitle	:= 'ST';
	pa_tyXMLTable[iTotalIdxWrite].sValue	:= 'ServiceDescription';
	pa_tyXMLTable[iTotalIdxWrite].uiSize	:= LEN(pa_tyXMLTable[iTotalIdxWrite].sValue);

	iTotalIdxWrite	:= iTotalIdxWrite + 1;

	IF tyParameter.tyAvl.bLaneId = TRUE THEN
		pa_tyXMLTable[iTotalIdxWrite].sTitle	:= 'AT';
		pa_tyXMLTable[iTotalIdxWrite].sValue	:= 'LaneId';
		pa_tyXMLTable[iTotalIdxWrite].uiSize	:= LEN(pa_tyXMLTable[iTotalIdxWrite].sValue);

		iTotalIdxWrite	:= iTotalIdxWrite + 1;

		pa_tyXMLTable[iTotalIdxWrite].sTitle	:= 'AV';
		pa_tyXMLTable[iTotalIdxWrite].sValue	:= INT_TO_STRING(tyParameter.tyData.iLaneId);
		pa_tyXMLTable[iTotalIdxWrite].uiSize	:= LEN(pa_tyXMLTable[iTotalIdxWrite].sValue);

		iTotalIdxWrite	:= iTotalIdxWrite + 1;
	END_IF

	IF tyParameter.tyAvl.bMachineId = TRUE THEN
		pa_tyXMLTable[iTotalIdxWrite].sTitle	:= 'AT';
		pa_tyXMLTable[iTotalIdxWrite].sValue	:= 'MachineId';
		pa_tyXMLTable[iTotalIdxWrite].uiSize	:= LEN(pa_tyXMLTable[iTotalIdxWrite].sValue);

		iTotalIdxWrite	:= iTotalIdxWrite + 1;

		pa_tyXMLTable[iTotalIdxWrite].sTitle	:= 'AV';
		pa_tyXMLTable[iTotalIdxWrite].sValue	:= tyParameter.tyData.sMachineId;
		pa_tyXMLTable[iTotalIdxWrite].uiSize	:= LEN(pa_tyXMLTable[iTotalIdxWrite].sValue);

		iTotalIdxWrite	:= iTotalIdxWrite + 1;
	END_IF

	IF tyParameter.tyAvl.bInterfaceId = TRUE THEN
		pa_tyXMLTable[iTotalIdxWrite].sTitle	:= 'AT';
		pa_tyXMLTable[iTotalIdxWrite].sValue	:= 'InterfaceId';
		pa_tyXMLTable[iTotalIdxWrite].uiSize	:= LEN(pa_tyXMLTable[iTotalIdxWrite].sValue);

		iTotalIdxWrite	:= iTotalIdxWrite + 1;

		pa_tyXMLTable[iTotalIdxWrite].sTitle	:= 'AV';
		pa_tyXMLTable[iTotalIdxWrite].sValue	:= tyParameter.tyData.sInterfaceId;
		pa_tyXMLTable[iTotalIdxWrite].uiSize	:= LEN(pa_tyXMLTable[iTotalIdxWrite].sValue);

		iTotalIdxWrite	:= iTotalIdxWrite + 1;
	END_IF

	IF tyParameter.tyAvl.bVersion = TRUE THEN
		pa_tyXMLTable[iTotalIdxWrite].sTitle	:= 'AT';
		pa_tyXMLTable[iTotalIdxWrite].sValue	:= 'Version';
		pa_tyXMLTable[iTotalIdxWrite].uiSize	:= LEN(pa_tyXMLTable[iTotalIdxWrite].sValue);

		iTotalIdxWrite	:= iTotalIdxWrite + 1;

		pa_tyXMLTable[iTotalIdxWrite].sTitle	:= 'AV';
		pa_tyXMLTable[iTotalIdxWrite].sValue	:= tyParameter.tyData.sVersion;
		pa_tyXMLTable[iTotalIdxWrite].uiSize	:= LEN(pa_tyXMLTable[iTotalIdxWrite].sValue);

		iTotalIdxWrite	:= iTotalIdxWrite + 1;
	END_IF

	pa_tyXMLTable[iTotalIdxWrite].sTitle	:= 'EN';
	pa_tyXMLTable[iTotalIdxWrite].sValue	:= '';
	pa_tyXMLTable[iTotalIdxWrite].uiSize	:= LEN(pa_tyXMLTable[iTotalIdxWrite].sValue);

	iTotalIdxWrite	:= iTotalIdxWrite + 1;

	pa_tyXMLTable[iTotalIdxWrite].sTitle	:= 'ST';
	pa_tyXMLTable[iTotalIdxWrite].sValue	:= 'SupportedFeatures';
	pa_tyXMLTable[iTotalIdxWrite].uiSize	:= LEN(pa_tyXMLTable[iTotalIdxWrite].sValue);

	iTotalIdxWrite	:= iTotalIdxWrite + 1;

	IF tyParameter.tyAvl.tySupportedFeatures.bFeatureBoardForecast = TRUE OR tyParameter.tyAvl.tySupportedFeatures.bFeatureCheckAliveResponse = TRUE OR tyParameter.tyAvl.tySupportedFeatures.bFeatureQueryBoardInfo = TRUE OR tyParameter.tyAvl.tySupportedFeatures.bFeatureSendBoardInfo = TRUE OR tyParameter.tyAvl.tySupportedFeatures.bFeatureCommand = TRUE THEN

		pa_tyXMLTable[iTotalIdxWrite].sTitle	:= 'EN';
		pa_tyXMLTable[iTotalIdxWrite].sValue	:= '';
		pa_tyXMLTable[iTotalIdxWrite].uiSize	:= LEN(pa_tyXMLTable[iTotalIdxWrite].sValue);

		iTotalIdxWrite	:= iTotalIdxWrite + 1;

		IF tyParameter.tyAvl.tySupportedFeatures.bFeatureBoardForecast = TRUE THEN
			pa_tyXMLTable[iTotalIdxWrite].sTitle	:= 'ST';
			pa_tyXMLTable[iTotalIdxWrite].sValue	:= 'FeatureBoardForecast';
			pa_tyXMLTable[iTotalIdxWrite].uiSize	:= LEN(pa_tyXMLTable[iTotalIdxWrite].sValue);

			iTotalIdxWrite	:= iTotalIdxWrite + 1;

			pa_tyXMLTable[iTotalIdxWrite].sTitle	:= 'ES';
			pa_tyXMLTable[iTotalIdxWrite].sValue	:= '';
			pa_tyXMLTable[iTotalIdxWrite].uiSize	:= LEN(pa_tyXMLTable[iTotalIdxWrite].sValue);

			iTotalIdxWrite	:= iTotalIdxWrite + 1;
		END_IF

		IF tyParameter.tyAvl.tySupportedFeatures.bFeatureCheckAliveResponse = TRUE THEN
			pa_tyXMLTable[iTotalIdxWrite].sTitle	:= 'ST';
			pa_tyXMLTable[iTotalIdxWrite].sValue	:= 'FeatureCheckAliveResponse';
			pa_tyXMLTable[iTotalIdxWrite].uiSize	:= LEN(pa_tyXMLTable[iTotalIdxWrite].sValue);

			iTotalIdxWrite	:= iTotalIdxWrite + 1;

			pa_tyXMLTable[iTotalIdxWrite].sTitle	:= 'ES';
			pa_tyXMLTable[iTotalIdxWrite].sValue	:= '';
			pa_tyXMLTable[iTotalIdxWrite].uiSize	:= LEN(pa_tyXMLTable[iTotalIdxWrite].sValue);

			iTotalIdxWrite	:= iTotalIdxWrite + 1;
		END_IF

		IF tyParameter.tyAvl.tySupportedFeatures.bFeatureQueryBoardInfo = TRUE THEN
			pa_tyXMLTable[iTotalIdxWrite].sTitle	:= 'ST';
			pa_tyXMLTable[iTotalIdxWrite].sValue	:= 'FeatureQueryBoardInfo';
			pa_tyXMLTable[iTotalIdxWrite].uiSize	:= LEN(pa_tyXMLTable[iTotalIdxWrite].sValue);

			iTotalIdxWrite	:= iTotalIdxWrite + 1;

			pa_tyXMLTable[iTotalIdxWrite].sTitle	:= 'ES';
			pa_tyXMLTable[iTotalIdxWrite].sValue	:= '';
			pa_tyXMLTable[iTotalIdxWrite].uiSize	:= LEN(pa_tyXMLTable[iTotalIdxWrite].sValue);

			iTotalIdxWrite	:= iTotalIdxWrite + 1;
		END_IF

		IF tyParameter.tyAvl.tySupportedFeatures.bFeatureSendBoardInfo = TRUE THEN
			pa_tyXMLTable[iTotalIdxWrite].sTitle	:= 'ST';
			pa_tyXMLTable[iTotalIdxWrite].sValue	:= 'FeatureSendBoardInfo';
			pa_tyXMLTable[iTotalIdxWrite].uiSize	:= LEN(pa_tyXMLTable[iTotalIdxWrite].sValue);

			iTotalIdxWrite	:= iTotalIdxWrite + 1;

			pa_tyXMLTable[iTotalIdxWrite].sTitle	:= 'ES';
			pa_tyXMLTable[iTotalIdxWrite].sValue	:= '';
			pa_tyXMLTable[iTotalIdxWrite].uiSize	:= LEN(pa_tyXMLTable[iTotalIdxWrite].sValue);

			iTotalIdxWrite	:= iTotalIdxWrite + 1;
		END_IF

		IF tyParameter.tyAvl.tySupportedFeatures.bFeatureCommand = TRUE  THEN
			pa_tyXMLTable[iTotalIdxWrite].sTitle	:= 'ST';
			pa_tyXMLTable[iTotalIdxWrite].sValue	:= 'FeatureCommand';
			pa_tyXMLTable[iTotalIdxWrite].uiSize	:= LEN(pa_tyXMLTable[iTotalIdxWrite].sValue);

			iTotalIdxWrite	:= iTotalIdxWrite + 1;

			pa_tyXMLTable[iTotalIdxWrite].sTitle	:= 'ES';
			pa_tyXMLTable[iTotalIdxWrite].sValue	:= '';
			pa_tyXMLTable[iTotalIdxWrite].uiSize	:= LEN(pa_tyXMLTable[iTotalIdxWrite].sValue);

			iTotalIdxWrite	:= iTotalIdxWrite + 1;

		END_IF

		pa_tyXMLTable[iTotalIdxWrite].sTitle	:= 'ET';
		pa_tyXMLTable[iTotalIdxWrite].sValue	:= 'SupportedFeatures';
		pa_tyXMLTable[iTotalIdxWrite].uiSize	:= LEN(pa_tyXMLTable[iTotalIdxWrite].sValue);

		iTotalIdxWrite	:= iTotalIdxWrite + 1;

		pa_tyXMLTable[iTotalIdxWrite].sTitle	:= 'EN';
		pa_tyXMLTable[iTotalIdxWrite].sValue	:= '';
		pa_tyXMLTable[iTotalIdxWrite].uiSize	:= LEN(pa_tyXMLTable[iTotalIdxWrite].sValue);

		iTotalIdxWrite	:= iTotalIdxWrite + 1;

	ELSE
		pa_tyXMLTable[iTotalIdxWrite].sTitle	:= 'ES';
		pa_tyXMLTable[iTotalIdxWrite].sValue	:= '';
		pa_tyXMLTable[iTotalIdxWrite].uiSize	:= LEN(pa_tyXMLTable[iTotalIdxWrite].sValue);

		iTotalIdxWrite	:= iTotalIdxWrite + 1;
	END_IF

	pa_tyXMLTable[iTotalIdxWrite].sTitle	:= 'ET';
	pa_tyXMLTable[iTotalIdxWrite].sValue	:= 'ServiceDescription';
	pa_tyXMLTable[iTotalIdxWrite].uiSize	:= LEN(pa_tyXMLTable[iTotalIdxWrite].sValue);

	iTotalIdxWrite	:= iTotalIdxWrite + 1;

	pa_tyXMLTable[iTotalIdxWrite].sTitle	:= 'EN';
	pa_tyXMLTable[iTotalIdxWrite].sValue	:= '';
	pa_tyXMLTable[iTotalIdxWrite].uiSize	:= LEN(pa_tyXMLTable[iTotalIdxWrite].sValue);

	iTotalIdxWrite	:= iTotalIdxWrite + 1;

	pa_tyXMLTable[iTotalIdxWrite].sTitle	:= 'ET';
	pa_tyXMLTable[iTotalIdxWrite].sValue	:= 'Hermes';
	pa_tyXMLTable[iTotalIdxWrite].uiSize	:= LEN(pa_tyXMLTable[iTotalIdxWrite].sValue);

	iTotalIdxWrite	:= iTotalIdxWrite + 1;

	pa_tyXMLTable[iTotalIdxWrite].sTitle	:= 'EN';
	pa_tyXMLTable[iTotalIdxWrite].sValue	:= '';
	pa_tyXMLTable[iTotalIdxWrite].uiSize	:= LEN(pa_tyXMLTable[iTotalIdxWrite].sValue);

	iTotalIdxWrite	:= iTotalIdxWrite + 1;

	iTotalIdxWrite	:= fHermesFormServiceDescription;

END_FUNCTION
```

#### fHermesFormSServiceDescription.st
```iecst
(* Hermes Form Service Description Table Data (Total Index Written In Table) *)
FUNCTION fHermesFormSServiceDescription

	memset(ADR(pa_tyXMLTable) , 0 , SIZEOF(pa_tyXMLTable));
	iTotalIdxWrite	:= 0;

	fHermesGetTimestamp(ADR(sTimestamp) , tyDTStructure);

	pa_tyXMLTable[iTotalIdxWrite].sTitle	:= 'ST';
	pa_tyXMLTable[iTotalIdxWrite].sValue	:= 'Hermes';
	pa_tyXMLTable[iTotalIdxWrite].uiSize	:= LEN(pa_tyXMLTable[iTotalIdxWrite].sValue);

	iTotalIdxWrite	:= iTotalIdxWrite + 1;

	pa_tyXMLTable[iTotalIdxWrite].sTitle	:= 'AT';
	pa_tyXMLTable[iTotalIdxWrite].sValue	:= 'Timestamp';
	pa_tyXMLTable[iTotalIdxWrite].uiSize	:= LEN(pa_tyXMLTable[iTotalIdxWrite].sValue);

	iTotalIdxWrite	:= iTotalIdxWrite + 1;

	pa_tyXMLTable[iTotalIdxWrite].sTitle	:= 'AV';
	pa_tyXMLTable[iTotalIdxWrite].sValue	:= sTimestamp;
	pa_tyXMLTable[iTotalIdxWrite].uiSize	:= LEN(pa_tyXMLTable[iTotalIdxWrite].sValue);

	iTotalIdxWrite	:= iTotalIdxWrite + 1;

	pa_tyXMLTable[iTotalIdxWrite].sTitle	:= 'EN';
	pa_tyXMLTable[iTotalIdxWrite].sValue	:= '';
	pa_tyXMLTable[iTotalIdxWrite].uiSize	:= LEN(pa_tyXMLTable[iTotalIdxWrite].sValue);

	iTotalIdxWrite	:= iTotalIdxWrite + 1;

	pa_tyXMLTable[iTotalIdxWrite].sTitle	:= 'ST';
	pa_tyXMLTable[iTotalIdxWrite].sValue	:= 'SupervisoryServiceDescription';
	pa_tyXMLTable[iTotalIdxWrite].uiSize	:= LEN(pa_tyXMLTable[iTotalIdxWrite].sValue);

	iTotalIdxWrite	:= iTotalIdxWrite + 1;

	IF tyParameter.tyAvl.bSystemId = TRUE THEN
		pa_tyXMLTable[iTotalIdxWrite].sTitle	:= 'AT';
		pa_tyXMLTable[iTotalIdxWrite].sValue	:= 'SystemId';
		pa_tyXMLTable[iTotalIdxWrite].uiSize	:= LEN(pa_tyXMLTable[iTotalIdxWrite].sValue);

		iTotalIdxWrite	:= iTotalIdxWrite + 1;

		pa_tyXMLTable[iTotalIdxWrite].sTitle	:= 'AV';
		pa_tyXMLTable[iTotalIdxWrite].sValue	:= tyParameter.tyData.sSystemId;
		pa_tyXMLTable[iTotalIdxWrite].uiSize	:= LEN(pa_tyXMLTable[iTotalIdxWrite].sValue);

		iTotalIdxWrite	:= iTotalIdxWrite + 1;
	END_IF

	IF tyParameter.tyAvl.bVersion = TRUE THEN
		pa_tyXMLTable[iTotalIdxWrite].sTitle	:= 'AT';
		pa_tyXMLTable[iTotalIdxWrite].sValue	:= 'Version';
		pa_tyXMLTable[iTotalIdxWrite].uiSize	:= LEN(pa_tyXMLTable[iTotalIdxWrite].sValue);

		iTotalIdxWrite	:= iTotalIdxWrite + 1;

		pa_tyXMLTable[iTotalIdxWrite].sTitle	:= 'AV';
		pa_tyXMLTable[iTotalIdxWrite].sValue	:= tyParameter.tyData.sVersion;
		pa_tyXMLTable[iTotalIdxWrite].uiSize	:= LEN(pa_tyXMLTable[iTotalIdxWrite].sValue);

		iTotalIdxWrite	:= iTotalIdxWrite + 1;
	END_IF

	pa_tyXMLTable[iTotalIdxWrite].sTitle	:= 'EN';
	pa_tyXMLTable[iTotalIdxWrite].sValue	:= '';
	pa_tyXMLTable[iTotalIdxWrite].uiSize	:= LEN(pa_tyXMLTable[iTotalIdxWrite].sValue);

	iTotalIdxWrite	:= iTotalIdxWrite + 1;

	pa_tyXMLTable[iTotalIdxWrite].sTitle	:= 'ST';
	pa_tyXMLTable[iTotalIdxWrite].sValue	:= 'SupportedFeatures';
	pa_tyXMLTable[iTotalIdxWrite].uiSize	:= LEN(pa_tyXMLTable[iTotalIdxWrite].sValue);

	iTotalIdxWrite	:= iTotalIdxWrite + 1;

	IF tyParameter.tyAvl.tySupportedFeatures.bFeatureConfiguration = TRUE OR tyParameter.tyAvl.tySupportedFeatures.bFeatureCheckAliveResponse = TRUE OR tyParameter.tyAvl.tySupportedFeatures.bFeatureBoardTracking = TRUE OR tyParameter.tyAvl.tySupportedFeatures.bFeatureQueryWorkOrderInfo = TRUE OR tyParameter.tyAvl.tySupportedFeatures.bFeatureSendWorkOrderInfo = TRUE THEN

		pa_tyXMLTable[iTotalIdxWrite].sTitle	:= 'EN';
		pa_tyXMLTable[iTotalIdxWrite].sValue	:= '';
		pa_tyXMLTable[iTotalIdxWrite].uiSize	:= LEN(pa_tyXMLTable[iTotalIdxWrite].sValue);

		iTotalIdxWrite	:= iTotalIdxWrite + 1;

		IF tyParameter.tyAvl.tySupportedFeatures.bFeatureConfiguration = TRUE THEN
			pa_tyXMLTable[iTotalIdxWrite].sTitle	:= 'ST';
			pa_tyXMLTable[iTotalIdxWrite].sValue	:= 'FeatureConfiguration';
			pa_tyXMLTable[iTotalIdxWrite].uiSize	:= LEN(pa_tyXMLTable[iTotalIdxWrite].sValue);

			iTotalIdxWrite	:= iTotalIdxWrite + 1;

			pa_tyXMLTable[iTotalIdxWrite].sTitle	:= 'ES';
			pa_tyXMLTable[iTotalIdxWrite].sValue	:= '';
			pa_tyXMLTable[iTotalIdxWrite].uiSize	:= LEN(pa_tyXMLTable[iTotalIdxWrite].sValue);

			iTotalIdxWrite	:= iTotalIdxWrite + 1;
		END_IF

		IF tyParameter.tyAvl.tySupportedFeatures.bFeatureCheckAliveResponse = TRUE THEN
			pa_tyXMLTable[iTotalIdxWrite].sTitle	:= 'ST';
			pa_tyXMLTable[iTotalIdxWrite].sValue	:= 'FeatureCheckAliveResponse';
			pa_tyXMLTable[iTotalIdxWrite].uiSize	:= LEN(pa_tyXMLTable[iTotalIdxWrite].sValue);

			iTotalIdxWrite	:= iTotalIdxWrite + 1;

			pa_tyXMLTable[iTotalIdxWrite].sTitle	:= 'ES';
			pa_tyXMLTable[iTotalIdxWrite].sValue	:= '';
			pa_tyXMLTable[iTotalIdxWrite].uiSize	:= LEN(pa_tyXMLTable[iTotalIdxWrite].sValue);

			iTotalIdxWrite	:= iTotalIdxWrite + 1;
		END_IF

		IF tyParameter.tyAvl.tySupportedFeatures.bFeatureBoardTracking = TRUE THEN
			pa_tyXMLTable[iTotalIdxWrite].sTitle	:= 'ST';
			pa_tyXMLTable[iTotalIdxWrite].sValue	:= 'FeatureBoardTracking';
			pa_tyXMLTable[iTotalIdxWrite].uiSize	:= LEN(pa_tyXMLTable[iTotalIdxWrite].sValue);

			iTotalIdxWrite	:= iTotalIdxWrite + 1;

			pa_tyXMLTable[iTotalIdxWrite].sTitle	:= 'ES';
			pa_tyXMLTable[iTotalIdxWrite].sValue	:= '';
			pa_tyXMLTable[iTotalIdxWrite].uiSize	:= LEN(pa_tyXMLTable[iTotalIdxWrite].sValue);

			iTotalIdxWrite	:= iTotalIdxWrite + 1;
		END_IF

		IF tyParameter.tyAvl.tySupportedFeatures.bFeatureQueryWorkOrderInfo = TRUE THEN
			pa_tyXMLTable[iTotalIdxWrite].sTitle	:= 'ST';
			pa_tyXMLTable[iTotalIdxWrite].sValue	:= 'FeatureQueryWorkOrderInfo';
			pa_tyXMLTable[iTotalIdxWrite].uiSize	:= LEN(pa_tyXMLTable[iTotalIdxWrite].sValue);

			iTotalIdxWrite	:= iTotalIdxWrite + 1;

			pa_tyXMLTable[iTotalIdxWrite].sTitle	:= 'ES';
			pa_tyXMLTable[iTotalIdxWrite].sValue	:= '';
			pa_tyXMLTable[iTotalIdxWrite].uiSize	:= LEN(pa_tyXMLTable[iTotalIdxWrite].sValue);

			iTotalIdxWrite	:= iTotalIdxWrite + 1;
		END_IF

		IF tyParameter.tyAvl.tySupportedFeatures.bFeatureSendWorkOrderInfo = TRUE THEN
			pa_tyXMLTable[iTotalIdxWrite].sTitle	:= 'ST';
			pa_tyXMLTable[iTotalIdxWrite].sValue	:= 'FeatureSendWorkOrderInfo';
			pa_tyXMLTable[iTotalIdxWrite].uiSize	:= LEN(pa_tyXMLTable[iTotalIdxWrite].sValue);

			iTotalIdxWrite	:= iTotalIdxWrite + 1;

			pa_tyXMLTable[iTotalIdxWrite].sTitle	:= 'ES';
			pa_tyXMLTable[iTotalIdxWrite].sValue	:= '';
			pa_tyXMLTable[iTotalIdxWrite].uiSize	:= LEN(pa_tyXMLTable[iTotalIdxWrite].sValue);

			iTotalIdxWrite	:= iTotalIdxWrite + 1;
		END_IF

		pa_tyXMLTable[iTotalIdxWrite].sTitle	:= 'ET';
		pa_tyXMLTable[iTotalIdxWrite].sValue	:= 'SupportedFeatures';
		pa_tyXMLTable[iTotalIdxWrite].uiSize	:= LEN(pa_tyXMLTable[iTotalIdxWrite].sValue);

		iTotalIdxWrite	:= iTotalIdxWrite + 1;

		pa_tyXMLTable[iTotalIdxWrite].sTitle	:= 'EN';
		pa_tyXMLTable[iTotalIdxWrite].sValue	:= '';
		pa_tyXMLTable[iTotalIdxWrite].uiSize	:= LEN(pa_tyXMLTable[iTotalIdxWrite].sValue);

		iTotalIdxWrite	:= iTotalIdxWrite + 1;

	ELSE
		pa_tyXMLTable[iTotalIdxWrite].sTitle	:= 'ES';
		pa_tyXMLTable[iTotalIdxWrite].sValue	:= '';
		pa_tyXMLTable[iTotalIdxWrite].uiSize	:= LEN(pa_tyXMLTable[iTotalIdxWrite].sValue);

		iTotalIdxWrite	:= iTotalIdxWrite + 1;
	END_IF

	pa_tyXMLTable[iTotalIdxWrite].sTitle	:= 'ET';
	pa_tyXMLTable[iTotalIdxWrite].sValue	:= 'SupervisoryServiceDescription';
	pa_tyXMLTable[iTotalIdxWrite].uiSize	:= LEN(pa_tyXMLTable[iTotalIdxWrite].sValue);

	iTotalIdxWrite	:= iTotalIdxWrite + 1;

	pa_tyXMLTable[iTotalIdxWrite].sTitle	:= 'EN';
	pa_tyXMLTable[iTotalIdxWrite].sValue	:= '';
	pa_tyXMLTable[iTotalIdxWrite].uiSize	:= LEN(pa_tyXMLTable[iTotalIdxWrite].sValue);

	iTotalIdxWrite	:= iTotalIdxWrite + 1;

	pa_tyXMLTable[iTotalIdxWrite].sTitle	:= 'ET';
	pa_tyXMLTable[iTotalIdxWrite].sValue	:= 'Hermes';
	pa_tyXMLTable[iTotalIdxWrite].uiSize	:= LEN(pa_tyXMLTable[iTotalIdxWrite].sValue);

	iTotalIdxWrite	:= iTotalIdxWrite + 1;

	pa_tyXMLTable[iTotalIdxWrite].sTitle	:= 'EN';
	pa_tyXMLTable[iTotalIdxWrite].sValue	:= '';
	pa_tyXMLTable[iTotalIdxWrite].uiSize	:= LEN(pa_tyXMLTable[iTotalIdxWrite].sValue);

	iTotalIdxWrite	:= iTotalIdxWrite + 1;

	iTotalIdxWrite	:= fHermesFormSServiceDescription;

END_FUNCTION
```

#### fHermesFormNotification.st
```iecst
(* Hermes Form Notification Table Data (Total Index Written In Table) *)
FUNCTION fHermesFormNotification

	memset(ADR(pa_tyXMLTable) , 0 , SIZEOF(pa_tyXMLTable));
	iTotalIdxWrite	:= 0;

	fHermesGetTimestamp(ADR(sTimestamp) , tyDTStructure);

	pa_tyXMLTable[iTotalIdxWrite].sTitle	:= 'ST';
	pa_tyXMLTable[iTotalIdxWrite].sValue	:= 'Hermes';
	pa_tyXMLTable[iTotalIdxWrite].uiSize	:= LEN(pa_tyXMLTable[iTotalIdxWrite].sValue);

	iTotalIdxWrite	:= iTotalIdxWrite + 1;

	pa_tyXMLTable[iTotalIdxWrite].sTitle	:= 'AT';
	pa_tyXMLTable[iTotalIdxWrite].sValue	:= 'Timestamp';
	pa_tyXMLTable[iTotalIdxWrite].uiSize	:= LEN(pa_tyXMLTable[iTotalIdxWrite].sValue);

	iTotalIdxWrite	:= iTotalIdxWrite + 1;

	pa_tyXMLTable[iTotalIdxWrite].sTitle	:= 'AV';
	pa_tyXMLTable[iTotalIdxWrite].sValue	:= sTimestamp;
	pa_tyXMLTable[iTotalIdxWrite].uiSize	:= LEN(pa_tyXMLTable[iTotalIdxWrite].sValue);

	iTotalIdxWrite	:= iTotalIdxWrite + 1;

	pa_tyXMLTable[iTotalIdxWrite].sTitle	:= 'EN';
	pa_tyXMLTable[iTotalIdxWrite].sValue	:= '';
	pa_tyXMLTable[iTotalIdxWrite].uiSize	:= LEN(pa_tyXMLTable[iTotalIdxWrite].sValue);

	iTotalIdxWrite	:= iTotalIdxWrite + 1;

	pa_tyXMLTable[iTotalIdxWrite].sTitle	:= 'ST';
	pa_tyXMLTable[iTotalIdxWrite].sValue	:= 'Notification';
	pa_tyXMLTable[iTotalIdxWrite].uiSize	:= LEN(pa_tyXMLTable[iTotalIdxWrite].sValue);

	iTotalIdxWrite	:= iTotalIdxWrite + 1;

	IF tyParameter.tyAvl.bNotificationCode = TRUE THEN
		pa_tyXMLTable[iTotalIdxWrite].sTitle	:= 'AT';
		pa_tyXMLTable[iTotalIdxWrite].sValue	:= 'NotificationCode';
		pa_tyXMLTable[iTotalIdxWrite].uiSize	:= LEN(pa_tyXMLTable[iTotalIdxWrite].sValue);

		iTotalIdxWrite	:= iTotalIdxWrite + 1;

		pa_tyXMLTable[iTotalIdxWrite].sTitle	:= 'AV';
		pa_tyXMLTable[iTotalIdxWrite].sValue	:= INT_TO_STRING(tyParameter.tyData.iNotificationCode);
		pa_tyXMLTable[iTotalIdxWrite].uiSize	:= LEN(pa_tyXMLTable[iTotalIdxWrite].sValue);

		iTotalIdxWrite	:= iTotalIdxWrite + 1;
	END_IF

	IF tyParameter.tyAvl.bSeverity = TRUE THEN
		pa_tyXMLTable[iTotalIdxWrite].sTitle	:= 'AT';
		pa_tyXMLTable[iTotalIdxWrite].sValue	:= 'Severity';
		pa_tyXMLTable[iTotalIdxWrite].uiSize	:= LEN(pa_tyXMLTable[iTotalIdxWrite].sValue);

		iTotalIdxWrite	:= iTotalIdxWrite + 1;

		pa_tyXMLTable[iTotalIdxWrite].sTitle	:= 'AV';
		pa_tyXMLTable[iTotalIdxWrite].sValue	:= DINT_TO_STRING(UDINT_TO_DINT(tyParameter.tyData.eSeverity));
		pa_tyXMLTable[iTotalIdxWrite].uiSize	:= LEN(pa_tyXMLTable[iTotalIdxWrite].sValue);

		iTotalIdxWrite	:= iTotalIdxWrite + 1;
	END_IF

	IF tyParameter.tyAvl.bDescription = TRUE THEN
		pa_tyXMLTable[iTotalIdxWrite].sTitle	:= 'AT';
		pa_tyXMLTable[iTotalIdxWrite].sValue	:= 'Description';
		pa_tyXMLTable[iTotalIdxWrite].uiSize	:= LEN(pa_tyXMLTable[iTotalIdxWrite].sValue);

		iTotalIdxWrite	:= iTotalIdxWrite + 1;

		pa_tyXMLTable[iTotalIdxWrite].sTitle	:= 'AV';
		pa_tyXMLTable[iTotalIdxWrite].sValue	:= tyParameter.tyData.sDescription;
		pa_tyXMLTable[iTotalIdxWrite].uiSize	:= LEN(pa_tyXMLTable[iTotalIdxWrite].sValue);

		iTotalIdxWrite	:= iTotalIdxWrite + 1;
	END_IF

	pa_tyXMLTable[iTotalIdxWrite].sTitle	:= 'ES';
	pa_tyXMLTable[iTotalIdxWrite].sValue	:= '';
	pa_tyXMLTable[iTotalIdxWrite].uiSize	:= LEN(pa_tyXMLTable[iTotalIdxWrite].sValue);

	iTotalIdxWrite	:= iTotalIdxWrite + 1;

	pa_tyXMLTable[iTotalIdxWrite].sTitle	:= 'ET';
	pa_tyXMLTable[iTotalIdxWrite].sValue	:= 'Hermes';
	pa_tyXMLTable[iTotalIdxWrite].uiSize	:= LEN(pa_tyXMLTable[iTotalIdxWrite].sValue);

	iTotalIdxWrite	:= iTotalIdxWrite + 1;

	pa_tyXMLTable[iTotalIdxWrite].sTitle	:= 'EN';
	pa_tyXMLTable[iTotalIdxWrite].sValue	:= '';
	pa_tyXMLTable[iTotalIdxWrite].uiSize	:= LEN(pa_tyXMLTable[iTotalIdxWrite].sValue);

	iTotalIdxWrite	:= iTotalIdxWrite + 1;

	iTotalIdxWrite	:= fHermesFormNotification;

END_FUNCTION
```
